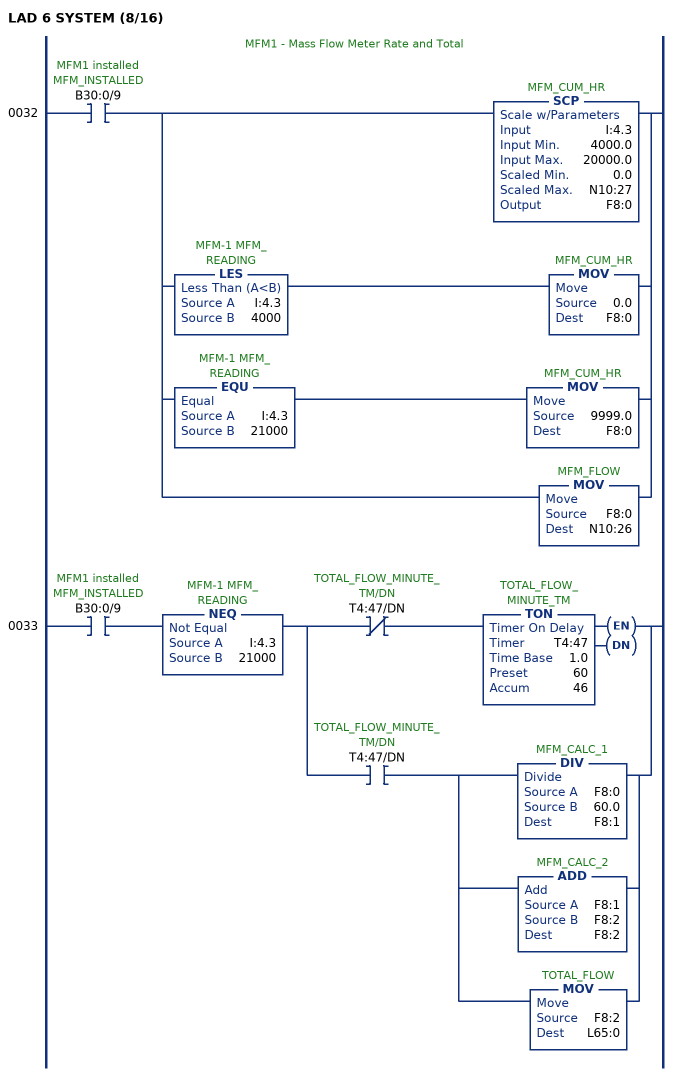
% Rung: 32 %
% MFM1 - Mass Flow Meter Rate and Total %
SOR XIC B30:0/9 BST SCP I:4.3 4000.0 20000.0 0.0 N10:27 F8:0 NXB LES I:4.3 4000 MOV 0.0 F8:0 NXB EQU I:4.3 21000 MOV 9999.0 F8:0 NXB MOV F8:0 N10:26 BND EOR
%   B30:0/9  MFM_INSTALLED  "MFM1 installed" %
%   I:4.3  MFM_READING  "MFM-1" %
%   N10:27  MFM_SCALING %
%   F8:0  MFM_CUM_HR %
%   N10:26  MFM_FLOW %
% Rung: 33 %
SOR XIC B30:0/9 NEQ I:4.3 21000 BST XIO T4:47/DN TON T4:47 1.0 60 46 NXB XIC T4:47/DN BST DIV F8:0 60.0 F8:1 NXB ADD F8:1 F8:2 F8:2 NXB MOV F8:2 L65:0 BND BND EOR
%   B30:0/9  MFM_INSTALLED  "MFM1 installed" %
%   I:4.3  MFM_READING  "MFM-1" %
%   T4:47  TOTAL_FLOW_MINUTE_TM %
%   F8:0  MFM_CUM_HR %
%   F8:1  MFM_CALC_1 %
%   F8:2  MFM_CALC_2 %
%   L65:0  TOTAL_FLOW %

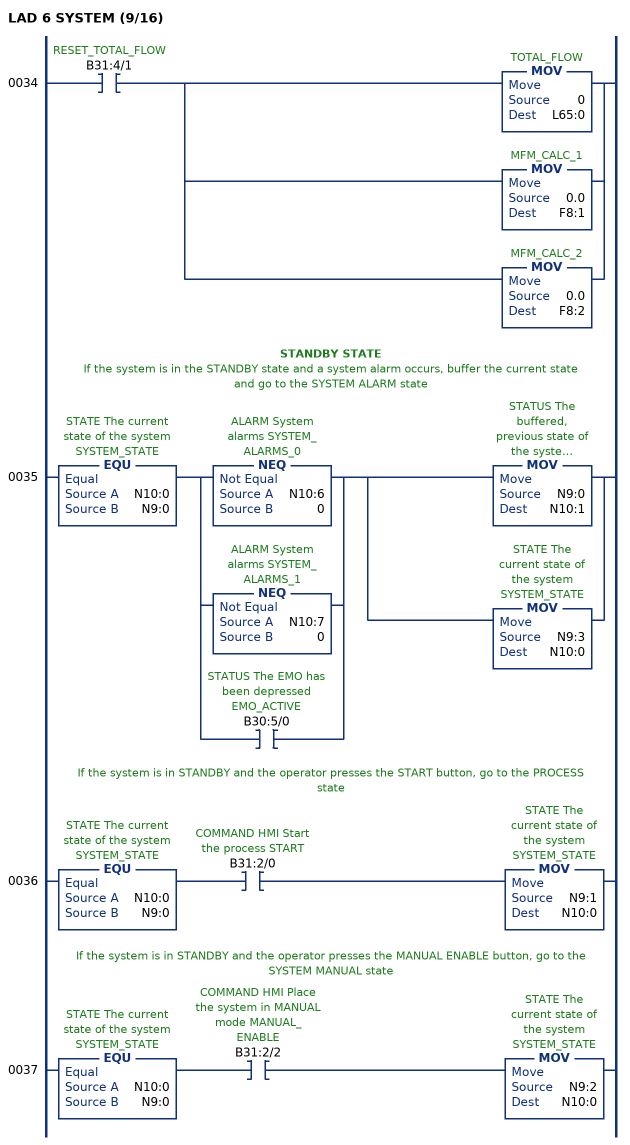
% Rung: 34 %
SOR XIC B31:4/1 BST MOV 0 L65:0 NXB MOV 0.0 F8:1 NXB MOV 0.0 F8:2 BND EOR
%   B31:4/1  RESET_TOTAL_FLOW %
%   L65:0  TOTAL_FLOW %
%   F8:1  MFM_CALC_1 %
%   F8:2  MFM_CALC_2 %
% Rung: 35 %
% TITLE: STANDBY STATE %
% If the system is in the STANDBY state and a system alarm occurs, buffer the current state and go to the SYSTEM ALARM state %
SOR EQU N10:0 N9:0 BST NEQ N10:6 0 NXB NEQ N10:7 0 NXB XIC B30:5/0 BND BST MOV N9:0 N10:1 NXB MOV N9:3 N10:0 BND EOR
%   N10:0  SYSTEM_STATE  "STATE The current state of the system" %
%   N9:0  SYSTEM_STANDBY  "STATE System Standby" %
%   N10:6  SYSTEM_ALARMS_0  "ALARM System alarms" %
%   N10:7  SYSTEM_ALARMS_1  "ALARM System alarms" %
%   B30:5/0  EMO_ACTIVE  "STATUS The EMO has been depressed" %
%   N10:1  SYSTEM_BUFFER  "STATUS The buffered, previous state of the system" %
%   N9:3  SYSTEM_ALARM  "STATE System Alarm" %
% Rung: 36 %
% If the system is in STANDBY and the operator presses the START button, go to the PROCESS state %
SOR EQU N10:0 N9:0 XIC B31:2/0 MOV N9:1 N10:0 EOR
%   N10:0  SYSTEM_STATE  "STATE The current state of the system" %
%   N9:0  SYSTEM_STANDBY  "STATE System Standby" %
%   B31:2/0  START  "COMMAND HMI Start the process" %
%   N9:1  SYSTEM_PROCESS  "STATE System Process" %
% Rung: 37 %
% If the system is in STANDBY and the operator presses the MANUAL ENABLE button, go to the SYSTEM MANUAL state %
SOR EQU N10:0 N9:0 XIC B31:2/2 MOV N9:2 N10:0 EOR
%   N10:0  SYSTEM_STATE  "STATE The current state of the system" %
%   N9:0  SYSTEM_STANDBY  "STATE System Standby" %
%   B31:2/2  MANUAL_ENABLE  "COMMAND HMI Place the system in MANUAL mode" %
%   N9:2  SYSTEM_MANUAL  "STATE System Manual" %

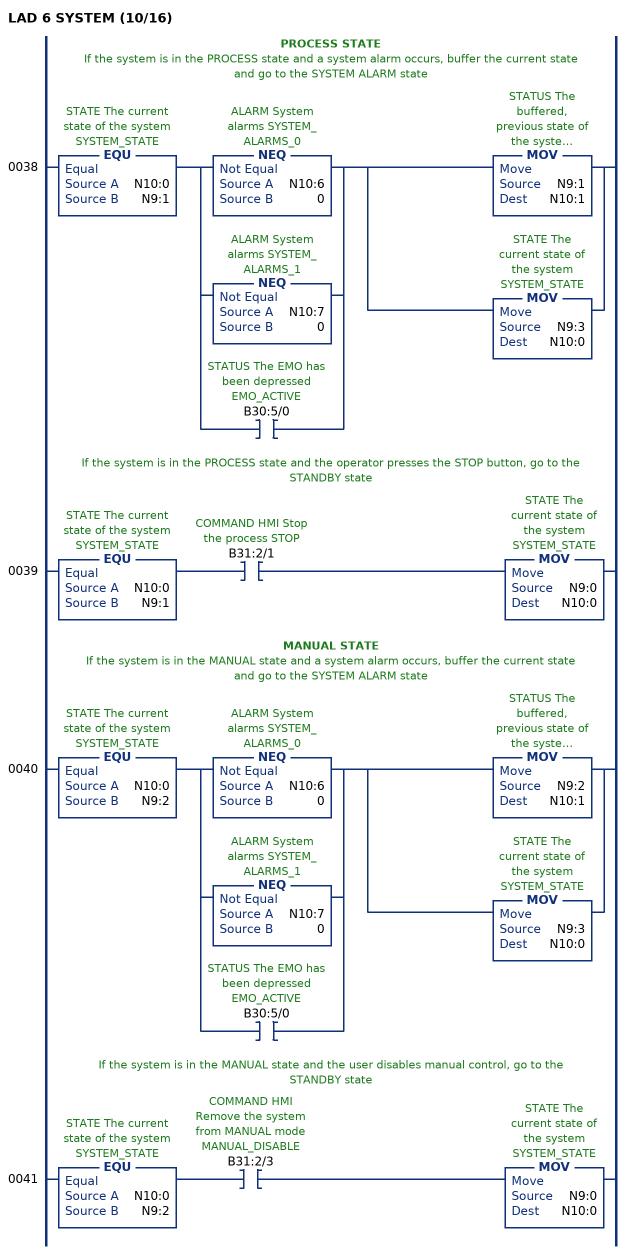
% Rung: 38 %
% TITLE: PROCESS STATE %
% If the system is in the PROCESS state and a system alarm occurs, buffer the current state and go to the SYSTEM ALARM state %
SOR EQU N10:0 N9:1 BST NEQ N10:6 0 NXB NEQ N10:7 0 NXB XIC B30:5/0 BND BST MOV N9:1 N10:1 NXB MOV N9:3 N10:0 BND EOR
%   N10:0  SYSTEM_STATE  "STATE The current state of the system" %
%   N9:1  SYSTEM_PROCESS  "STATE System Process" %
%   N10:6  SYSTEM_ALARMS_0  "ALARM System alarms" %
%   N10:7  SYSTEM_ALARMS_1  "ALARM System alarms" %
%   B30:5/0  EMO_ACTIVE  "STATUS The EMO has been depressed" %
%   N10:1  SYSTEM_BUFFER  "STATUS The buffered, previous state of the system" %
%   N9:3  SYSTEM_ALARM  "STATE System Alarm" %
% Rung: 39 %
% If the system is in the PROCESS state and the operator presses the STOP button, go to the STANDBY state %
SOR EQU N10:0 N9:1 XIC B31:2/1 MOV N9:0 N10:0 EOR
%   N10:0  SYSTEM_STATE  "STATE The current state of the system" %
%   N9:1  SYSTEM_PROCESS  "STATE System Process" %
%   B31:2/1  STOP  "COMMAND HMI Stop the process" %
%   N9:0  SYSTEM_STANDBY  "STATE System Standby" %
% Rung: 40 %
% TITLE: MANUAL STATE %
% If the system is in the MANUAL state and a system alarm occurs, buffer the current state and go to the SYSTEM ALARM state %
SOR EQU N10:0 N9:2 BST NEQ N10:6 0 NXB NEQ N10:7 0 NXB XIC B30:5/0 BND BST MOV N9:2 N10:1 NXB MOV N9:3 N10:0 BND EOR
%   N10:0  SYSTEM_STATE  "STATE The current state of the system" %
%   N9:2  SYSTEM_MANUAL  "STATE System Manual" %
%   N10:6  SYSTEM_ALARMS_0  "ALARM System alarms" %
%   N10:7  SYSTEM_ALARMS_1  "ALARM System alarms" %
%   B30:5/0  EMO_ACTIVE  "STATUS The EMO has been depressed" %
%   N10:1  SYSTEM_BUFFER  "STATUS The buffered, previous state of the system" %
%   N9:3  SYSTEM_ALARM  "STATE System Alarm" %
% Rung: 41 %
% If the system is in the MANUAL state and the user disables manual control, go to the STANDBY state %
SOR EQU N10:0 N9:2 XIC B31:2/3 MOV N9:0 N10:0 EOR
%   N10:0  SYSTEM_STATE  "STATE The current state of the system" %
%   N9:2  SYSTEM_MANUAL  "STATE System Manual" %
%   B31:2/3  MANUAL_DISABLE  "COMMAND HMI Remove the system from MANUAL mode" %
%   N9:0  SYSTEM_STANDBY  "STATE System Standby" %

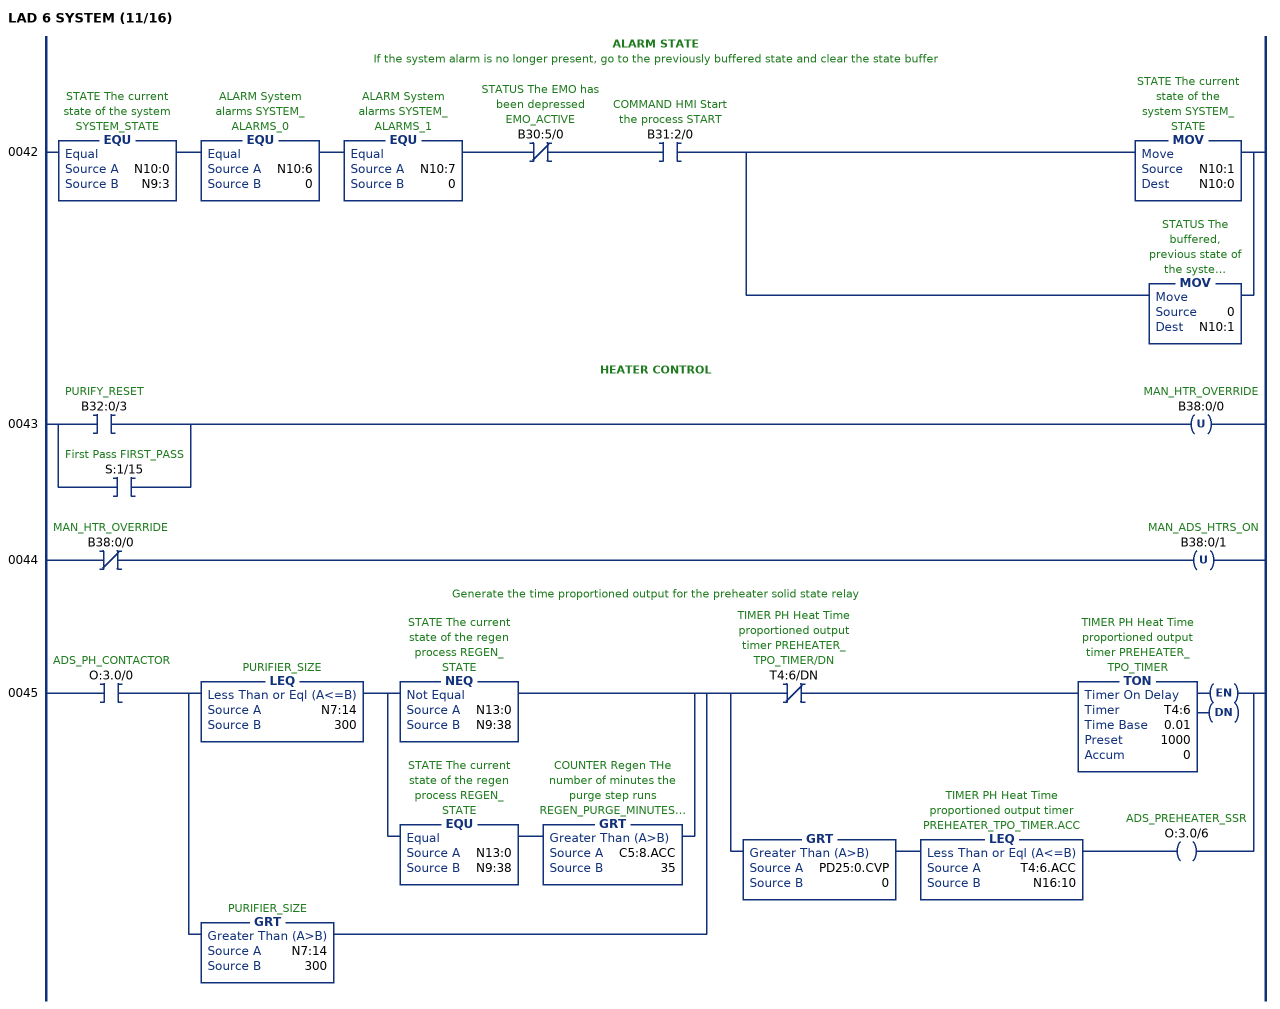
% Rung: 42 %
% TITLE: ALARM STATE %
% If the system alarm is no longer present, go to the previously buffered state and clear the state buffer %
SOR EQU N10:0 N9:3 EQU N10:6 0 EQU N10:7 0 XIO B30:5/0 XIC B31:2/0 BST MOV N10:1 N10:0 NXB MOV 0 N10:1 BND EOR
%   N10:0  SYSTEM_STATE  "STATE The current state of the system" %
%   N9:3  SYSTEM_ALARM  "STATE System Alarm" %
%   N10:6  SYSTEM_ALARMS_0  "ALARM System alarms" %
%   N10:7  SYSTEM_ALARMS_1  "ALARM System alarms" %
%   B30:5/0  EMO_ACTIVE  "STATUS The EMO has been depressed" %
%   B31:2/0  START  "COMMAND HMI Start the process" %
%   N10:1  SYSTEM_BUFFER  "STATUS The buffered, previous state of the system" %
% Rung: 43 %
% TITLE: HEATER CONTROL %
SOR BST XIC B32:0/3 NXB XIC S:1/15 BND OTU B38:0/0 EOR
%   B32:0/3  PURIFY_RESET %
%   S:1/15  FIRST_PASS  "First Pass" %
%   B38:0/0  MAN_HTR_OVERRIDE %
% Rung: 44 %
SOR XIO B38:0/0 OTU B38:0/1 EOR
%   B38:0/0  MAN_HTR_OVERRIDE %
%   B38:0/1  MAN_ADS_HTRS_ON %
% Rung: 45 %
% Generate the time proportioned output for the preheater solid state relay %
SOR XIC O:3.0/0 BST LEQ N7:14 300 BST NEQ N13:0 N9:38 NXB EQU N13:0 N9:38 GRT C5:8.ACC 35 BND NXB GRT N7:14 300 BND BST XIO T4:6/DN TON T4:6 0.01 1000 0 NXB GRT PD25:0.CVP 0 LEQ T4:6.ACC N16:10 OTE O:3.0/6 BND EOR
%   O:3.0/0  ADS_PH_CONTACTOR %
%   N7:14  PURIFIER_SIZE %
%   N13:0  REGEN_STATE  "STATE The current state of the regen process" %
%   N9:38  REGEN_PURGE  "STATE Regen Hot Purge" %
%   C5:8  REGEN_PURGE_MINUTES  "COUNTER Regen THe number of minutes the purge step runs" %
%   T4:6  PREHEATER_TPO_TIMER  "TIMER PH Heat Time proportioned output timer" %
%   N16:10  ADS_PH_OUTPUT  "CONTROL ADS Preheater output (percent)" %
%   O:3.0/6  ADS_PREHEATER_SSR %

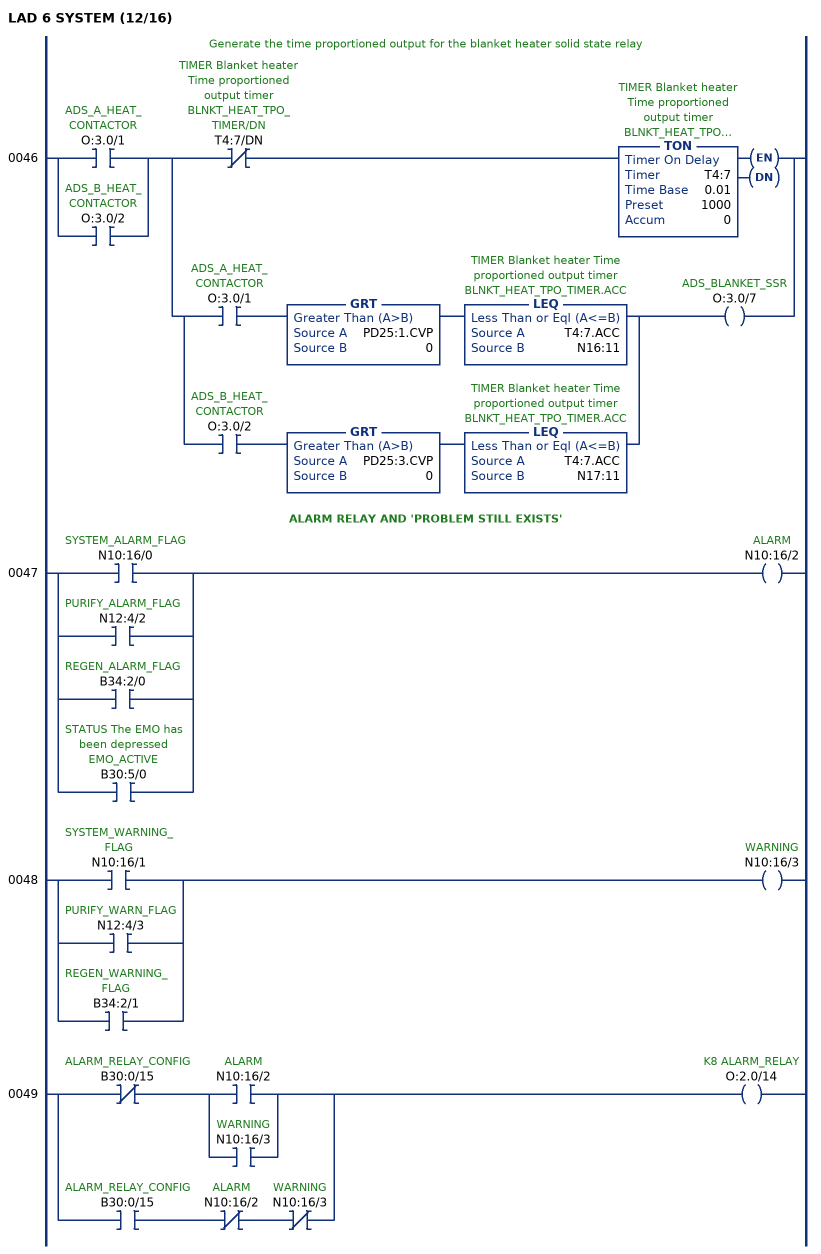
% Rung: 46 %
% Generate the time proportioned output for the blanket heater solid state relay %
SOR BST XIC O:3.0/1 NXB XIC O:3.0/2 BND BST XIO T4:7/DN TON T4:7 0.01 1000 0 NXB BST XIC O:3.0/1 GRT PD25:1.CVP 0 LEQ T4:7.ACC N16:11 NXB XIC O:3.0/2 GRT PD25:3.CVP 0 LEQ T4:7.ACC N17:11 BND OTE O:3.0/7 BND EOR
%   O:3.0/1  ADS_A_HEAT_CONTACTOR %
%   O:3.0/2  ADS_B_HEAT_CONTACTOR %
%   T4:7  BLNKT_HEAT_TPO_TIMER  "TIMER Blanket heater Time proportioned output timer" %
%   N16:11  ADS_A_BLNKT_OUTPUT  "CONTROL ADS A Blanket output (percent)" %
%   N17:11  ADS_B_BLNKT_OUTPUT  "CONTROL ADS A Blanket output" %
%   O:3.0/7  ADS_BLANKET_SSR %
% Rung: 47 %
% TITLE: ALARM RELAY AND 'PROBLEM STILL EXISTS' %
SOR BST XIC N10:16/0 NXB XIC N12:4/2 NXB XIC B34:2/0 NXB XIC B30:5/0 BND OTE N10:16/2 EOR
%   N10:16/0  SYSTEM_ALARM_FLAG %
%   N12:4/2  PURIFY_ALARM_FLAG %
%   B34:2/0  REGEN_ALARM_FLAG %
%   B30:5/0  EMO_ACTIVE  "STATUS The EMO has been depressed" %
%   N10:16/2  ALARM %
% Rung: 48 %
SOR BST XIC N10:16/1 NXB XIC N12:4/3 NXB XIC B34:2/1 BND OTE N10:16/3 EOR
%   N10:16/1  SYSTEM_WARNING_FLAG %
%   N12:4/3  PURIFY_WARN_FLAG %
%   B34:2/1  REGEN_WARNING_FLAG %
%   N10:16/3  WARNING %
% Rung: 49 %
SOR BST XIO B30:0/15 BST XIC N10:16/2 NXB XIC N10:16/3 BND NXB XIC B30:0/15 XIO N10:16/2 XIO N10:16/3 BND OTE O:2.0/14 EOR
%   B30:0/15  ALARM_RELAY_CONFIG %
%   N10:16/2  ALARM %
%   N10:16/3  WARNING %
%   O:2.0/14  ALARM_RELAY  "K8" %

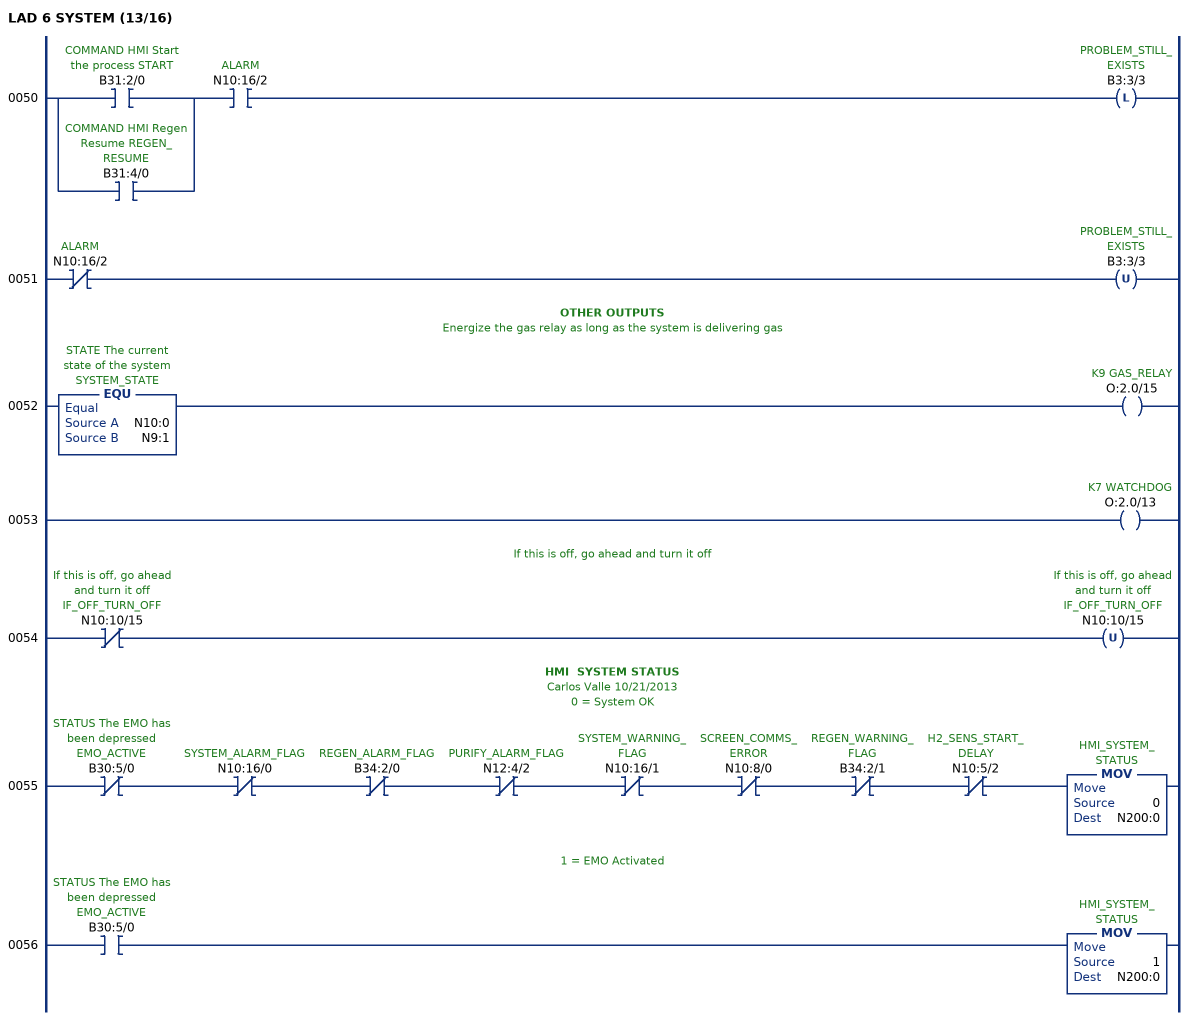
% Rung: 50 %
SOR BST XIC B31:2/0 NXB XIC B31:4/0 BND XIC N10:16/2 OTL B3:3/3 EOR
%   B31:2/0  START  "COMMAND HMI Start the process" %
%   B31:4/0  REGEN_RESUME  "COMMAND HMI Regen Resume" %
%   N10:16/2  ALARM %
%   B3:3/3  PROBLEM_STILL_EXISTS %
% Rung: 51 %
SOR XIO N10:16/2 OTU B3:3/3 EOR
%   N10:16/2  ALARM %
%   B3:3/3  PROBLEM_STILL_EXISTS %
% Rung: 52 %
% TITLE: OTHER OUTPUTS %
% Energize the gas relay as long as the system is delivering gas %
SOR EQU N10:0 N9:1 OTE O:2.0/15 EOR
%   N10:0  SYSTEM_STATE  "STATE The current state of the system" %
%   N9:1  SYSTEM_PROCESS  "STATE System Process" %
%   O:2.0/15  GAS_RELAY  "K9" %
% Rung: 53 %
SOR OTE O:2.0/13 EOR
%   O:2.0/13  WATCHDOG  "K7" %
% Rung: 54 %
% If this is off, go ahead and turn it off %
SOR XIO N10:10/15 OTU N10:10/15 EOR
%   N10:10/15  IF_OFF_TURN_OFF  "If this is off, go ahead and turn it off" %
% Rung: 55 %
% TITLE: HMI  SYSTEM STATUS %
% Carlos Valle 10/21/2013
% 0 = System OK %
SOR XIO B30:5/0 XIO N10:16/0 XIO B34:2/0 XIO N12:4/2 XIO N10:16/1 XIO N10:8/0 XIO B34:2/1 XIO N10:5/2 MOV 0 N200:0 EOR
%   B30:5/0  EMO_ACTIVE  "STATUS The EMO has been depressed" %
%   N10:16/0  SYSTEM_ALARM_FLAG %
%   B34:2/0  REGEN_ALARM_FLAG %
%   N12:4/2  PURIFY_ALARM_FLAG %
%   N10:16/1  SYSTEM_WARNING_FLAG %
%   N10:8/0  SCREEN_COMMS_ERROR %
%   B34:2/1  REGEN_WARNING_FLAG %
%   N10:5/2  H2_SENS_START_DELAY %
%   N200:0  HMI_SYSTEM_STATUS %
% Rung: 56 %
% 1 = EMO Activated %
SOR XIC B30:5/0 MOV 1 N200:0 EOR
%   B30:5/0  EMO_ACTIVE  "STATUS The EMO has been depressed" %
%   N200:0  HMI_SYSTEM_STATUS %

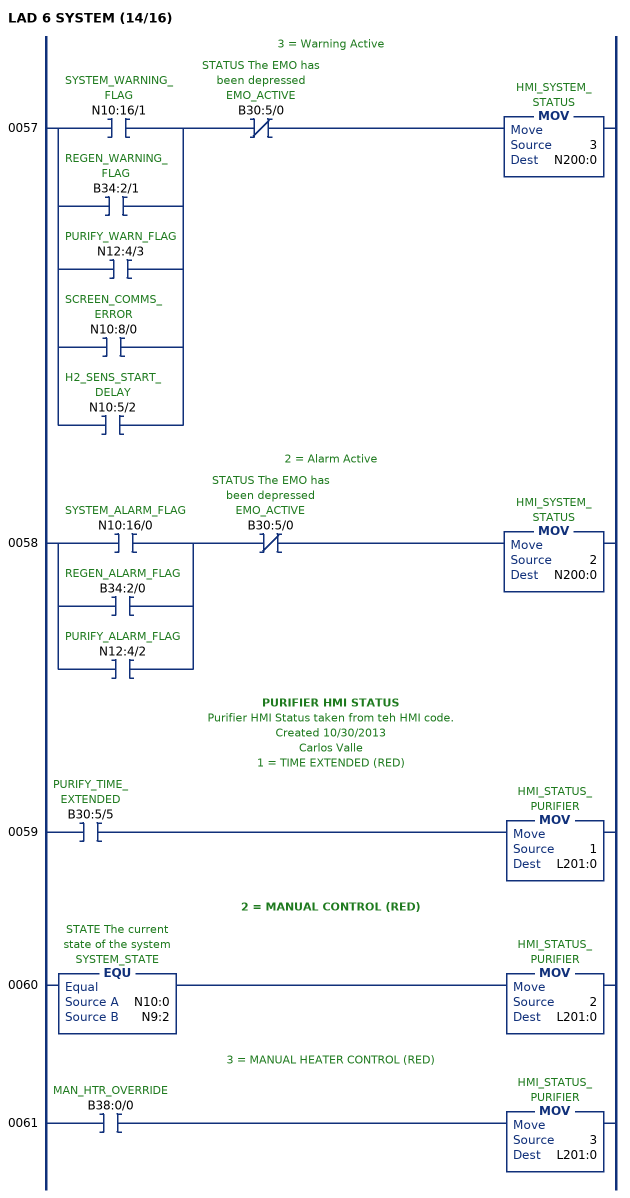
% Rung: 57 %
% 3 = Warning Active %
SOR BST XIC N10:16/1 NXB XIC B34:2/1 NXB XIC N12:4/3 NXB XIC N10:8/0 NXB XIC N10:5/2 BND XIO B30:5/0 MOV 3 N200:0 EOR
%   N10:16/1  SYSTEM_WARNING_FLAG %
%   B34:2/1  REGEN_WARNING_FLAG %
%   N12:4/3  PURIFY_WARN_FLAG %
%   N10:8/0  SCREEN_COMMS_ERROR %
%   N10:5/2  H2_SENS_START_DELAY %
%   B30:5/0  EMO_ACTIVE  "STATUS The EMO has been depressed" %
%   N200:0  HMI_SYSTEM_STATUS %
% Rung: 58 %
% 2 = Alarm Active %
SOR BST XIC N10:16/0 NXB XIC B34:2/0 NXB XIC N12:4/2 BND XIO B30:5/0 MOV 2 N200:0 EOR
%   N10:16/0  SYSTEM_ALARM_FLAG %
%   B34:2/0  REGEN_ALARM_FLAG %
%   N12:4/2  PURIFY_ALARM_FLAG %
%   B30:5/0  EMO_ACTIVE  "STATUS The EMO has been depressed" %
%   N200:0  HMI_SYSTEM_STATUS %
% Rung: 59 %
% TITLE: PURIFIER HMI STATUS %
% Purifier HMI Status taken from teh HMI code.
% Created 10/30/2013
% Carlos Valle
% 1 = TIME EXTENDED (RED) %
SOR XIC B30:5/5 MOV 1 L201:0 EOR
%   B30:5/5  PURIFY_TIME_EXTENDED %
%   L201:0  HMI_STATUS_PURIFIER %
% Rung: 60 %
% TITLE: 2 = MANUAL CONTROL (RED) %
SOR EQU N10:0 N9:2 MOV 2 L201:0 EOR
%   N10:0  SYSTEM_STATE  "STATE The current state of the system" %
%   N9:2  SYSTEM_MANUAL  "STATE System Manual" %
%   L201:0  HMI_STATUS_PURIFIER %
% Rung: 61 %
% 3 = MANUAL HEATER CONTROL (RED) %
SOR XIC B38:0/0 MOV 3 L201:0 EOR
%   B38:0/0  MAN_HTR_OVERRIDE %
%   L201:0  HMI_STATUS_PURIFIER %

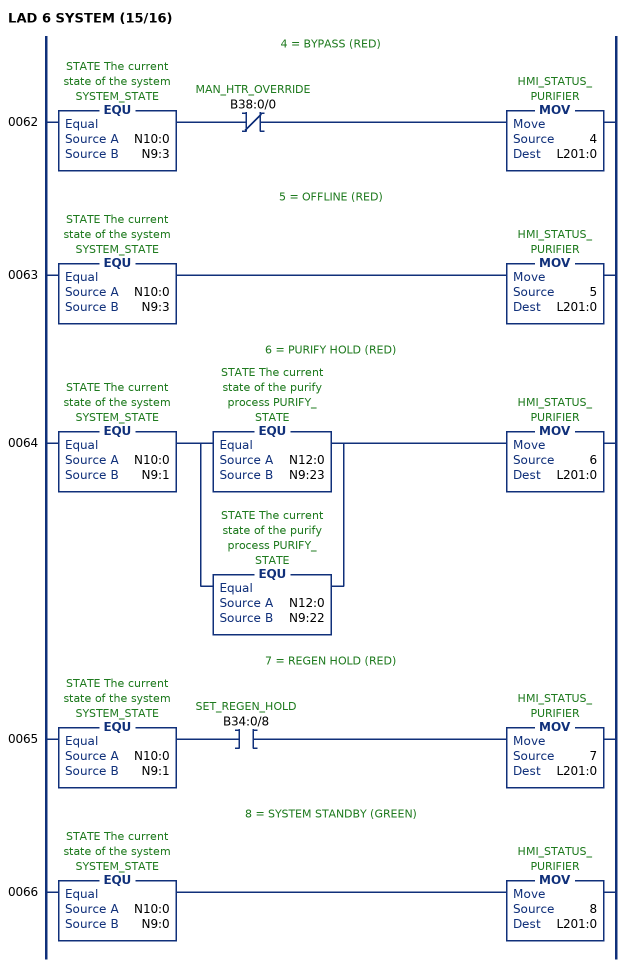
% Rung: 62 %
% 4 = BYPASS (RED) %
SOR EQU N10:0 N9:3 XIO B38:0/0 MOV 4 L201:0 EOR
%   N10:0  SYSTEM_STATE  "STATE The current state of the system" %
%   N9:3  SYSTEM_ALARM  "STATE System Alarm" %
%   B38:0/0  MAN_HTR_OVERRIDE %
%   L201:0  HMI_STATUS_PURIFIER %
% Rung: 63 %
% 5 = OFFLINE (RED) %
SOR EQU N10:0 N9:3 MOV 5 L201:0 EOR
%   N10:0  SYSTEM_STATE  "STATE The current state of the system" %
%   N9:3  SYSTEM_ALARM  "STATE System Alarm" %
%   L201:0  HMI_STATUS_PURIFIER %
% Rung: 64 %
% 6 = PURIFY HOLD (RED) %
SOR EQU N10:0 N9:1 BST EQU N12:0 N9:23 NXB EQU N12:0 N9:22 BND MOV 6 L201:0 EOR
%   N10:0  SYSTEM_STATE  "STATE The current state of the system" %
%   N9:1  SYSTEM_PROCESS  "STATE System Process" %
%   N12:0  PURIFY_STATE  "STATE The current state of the purify process" %
%   N9:23  PURIFY_MANUAL_HOLD  "STATE Purify Manual Hold" %
%   N9:22  PURIFY_HOLD  "STATE Purify Hold" %
%   L201:0  HMI_STATUS_PURIFIER %
% Rung: 65 %
% 7 = REGEN HOLD (RED) %
SOR EQU N10:0 N9:1 XIC B34:0/8 MOV 7 L201:0 EOR
%   N10:0  SYSTEM_STATE  "STATE The current state of the system" %
%   N9:1  SYSTEM_PROCESS  "STATE System Process" %
%   B34:0/8  SET_REGEN_HOLD %
%   L201:0  HMI_STATUS_PURIFIER %
% Rung: 66 %
% 8 = SYSTEM STANDBY (GREEN) %
SOR EQU N10:0 N9:0 MOV 8 L201:0 EOR
%   N10:0  SYSTEM_STATE  "STATE The current state of the system" %
%   N9:0  SYSTEM_STANDBY  "STATE System Standby" %
%   L201:0  HMI_STATUS_PURIFIER %

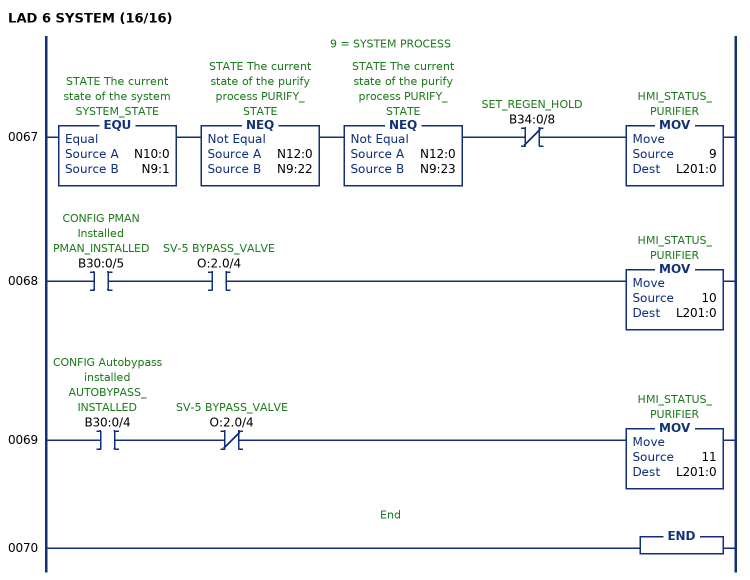
% Rung: 67 %
% 9 = SYSTEM PROCESS %
SOR EQU N10:0 N9:1 NEQ N12:0 N9:22 NEQ N12:0 N9:23 XIO B34:0/8 MOV 9 L201:0 EOR
%   N10:0  SYSTEM_STATE  "STATE The current state of the system" %
%   N9:1  SYSTEM_PROCESS  "STATE System Process" %
%   N12:0  PURIFY_STATE  "STATE The current state of the purify process" %
%   N9:22  PURIFY_HOLD  "STATE Purify Hold" %
%   N9:23  PURIFY_MANUAL_HOLD  "STATE Purify Manual Hold" %
%   B34:0/8  SET_REGEN_HOLD %
%   L201:0  HMI_STATUS_PURIFIER %
% Rung: 68 %
SOR XIC B30:0/5 XIC O:2.0/4 MOV 10 L201:0 EOR
%   B30:0/5  PMAN_INSTALLED  "CONFIG PMAN Installed" %
%   O:2.0/4  BYPASS_VALVE  "SV-5" %
%   L201:0  HMI_STATUS_PURIFIER %
% Rung: 69 %
SOR XIC B30:0/4 XIO O:2.0/4 MOV 11 L201:0 EOR
%   B30:0/4  AUTOBYPASS_INSTALLED  "CONFIG Autobypass installed" %
%   O:2.0/4  BYPASS_VALVE  "SV-5" %
%   L201:0  HMI_STATUS_PURIFIER %
% Rung: 70 %
% End %
SOR END EOR

LADDER 7 "PROCESSING"    % Runs the processing control %
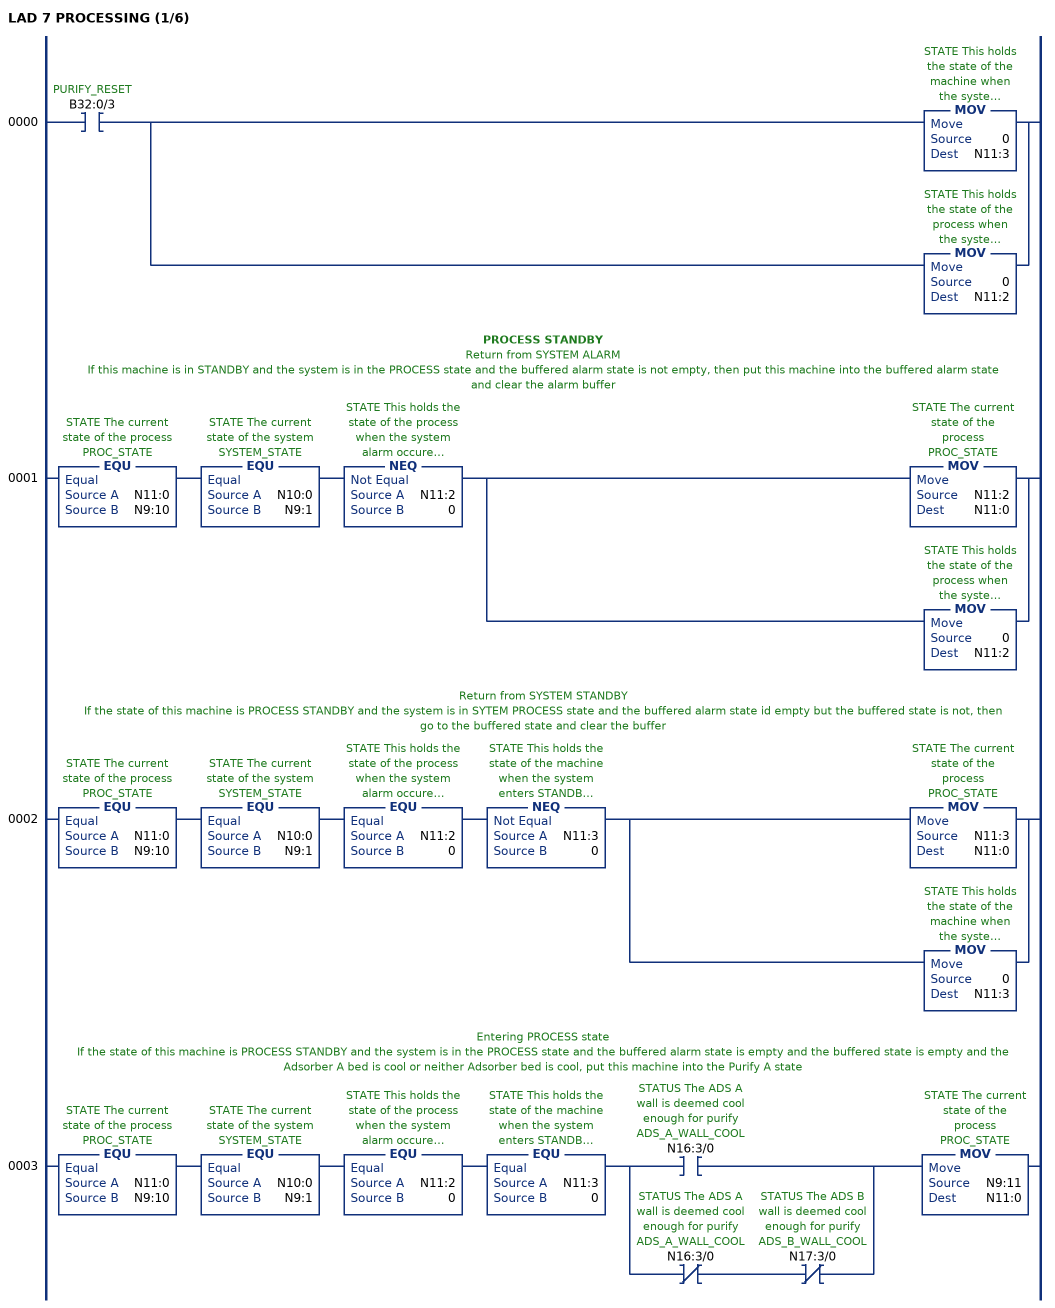
% Rung: 0 %
SOR XIC B32:0/3 BST MOV 0 N11:3 NXB MOV 0 N11:2 BND EOR
%   B32:0/3  PURIFY_RESET %
%   N11:3  PROC_STANDBY_BUFFER  "STATE This holds the state of the machine when the system enters STANDBY state" %
%   N11:2  PROC_ALARM_BUFFER  "STATE This holds the state of the process when the system alarm occured" %
% Rung: 1 %
% TITLE: PROCESS STANDBY %
% Return from SYSTEM ALARM
% If this machine is in STANDBY and the system is in the PROCESS state and the buffered alarm state is not empty, then put this machine into the buffered alarm state and clear the alarm buffer %
SOR EQU N11:0 N9:10 EQU N10:0 N9:1 NEQ N11:2 0 BST MOV N11:2 N11:0 NXB MOV 0 N11:2 BND EOR
%   N11:0  PROC_STATE  "STATE The current state of the process" %
%   N9:10  PROC_STANDBY  "STATE Process Standby" %
%   N10:0  SYSTEM_STATE  "STATE The current state of the system" %
%   N9:1  SYSTEM_PROCESS  "STATE System Process" %
%   N11:2  PROC_ALARM_BUFFER  "STATE This holds the state of the process when the system alarm occured" %
% Rung: 2 %
% Return from SYSTEM STANDBY
% If the state of this machine is PROCESS STANDBY and the system is in SYTEM PROCESS state and the buffered alarm state id empty but the buffered state is not, then go to the buffered state and clear the buffer %
SOR EQU N11:0 N9:10 EQU N10:0 N9:1 EQU N11:2 0 NEQ N11:3 0 BST MOV N11:3 N11:0 NXB MOV 0 N11:3 BND EOR
%   N11:0  PROC_STATE  "STATE The current state of the process" %
%   N9:10  PROC_STANDBY  "STATE Process Standby" %
%   N10:0  SYSTEM_STATE  "STATE The current state of the system" %
%   N9:1  SYSTEM_PROCESS  "STATE System Process" %
%   N11:2  PROC_ALARM_BUFFER  "STATE This holds the state of the process when the system alarm occured" %
%   N11:3  PROC_STANDBY_BUFFER  "STATE This holds the state of the machine when the system enters STANDBY state" %
% Rung: 3 %
% Entering PROCESS state
% If the state of this machine is PROCESS STANDBY and the system is in the PROCESS state and the buffered alarm state is empty and the buffered state is empty and the Adsorber A bed is cool or neither Adsorber bed is cool, put this machine into the Purify A state %
SOR EQU N11:0 N9:10 EQU N10:0 N9:1 EQU N11:2 0 EQU N11:3 0 BST XIC N16:3/0 NXB XIO N16:3/0 XIO N17:3/0 BND MOV N9:11 N11:0 EOR
%   N11:0  PROC_STATE  "STATE The current state of the process" %
%   N9:10  PROC_STANDBY  "STATE Process Standby" %
%   N10:0  SYSTEM_STATE  "STATE The current state of the system" %
%   N9:1  SYSTEM_PROCESS  "STATE System Process" %
%   N11:2  PROC_ALARM_BUFFER  "STATE This holds the state of the process when the system alarm occured" %
%   N11:3  PROC_STANDBY_BUFFER  "STATE This holds the state of the machine when the system enters STANDBY state" %
%   N16:3/0  ADS_A_WALL_COOL  "STATUS The ADS A wall is deemed cool enough for purify" %
%   N17:3/0  ADS_B_WALL_COOL  "STATUS The ADS B wall is deemed cool enough for purify" %
%   N9:11  PROC_PURIFY_A  "STATE Process Purify A" %

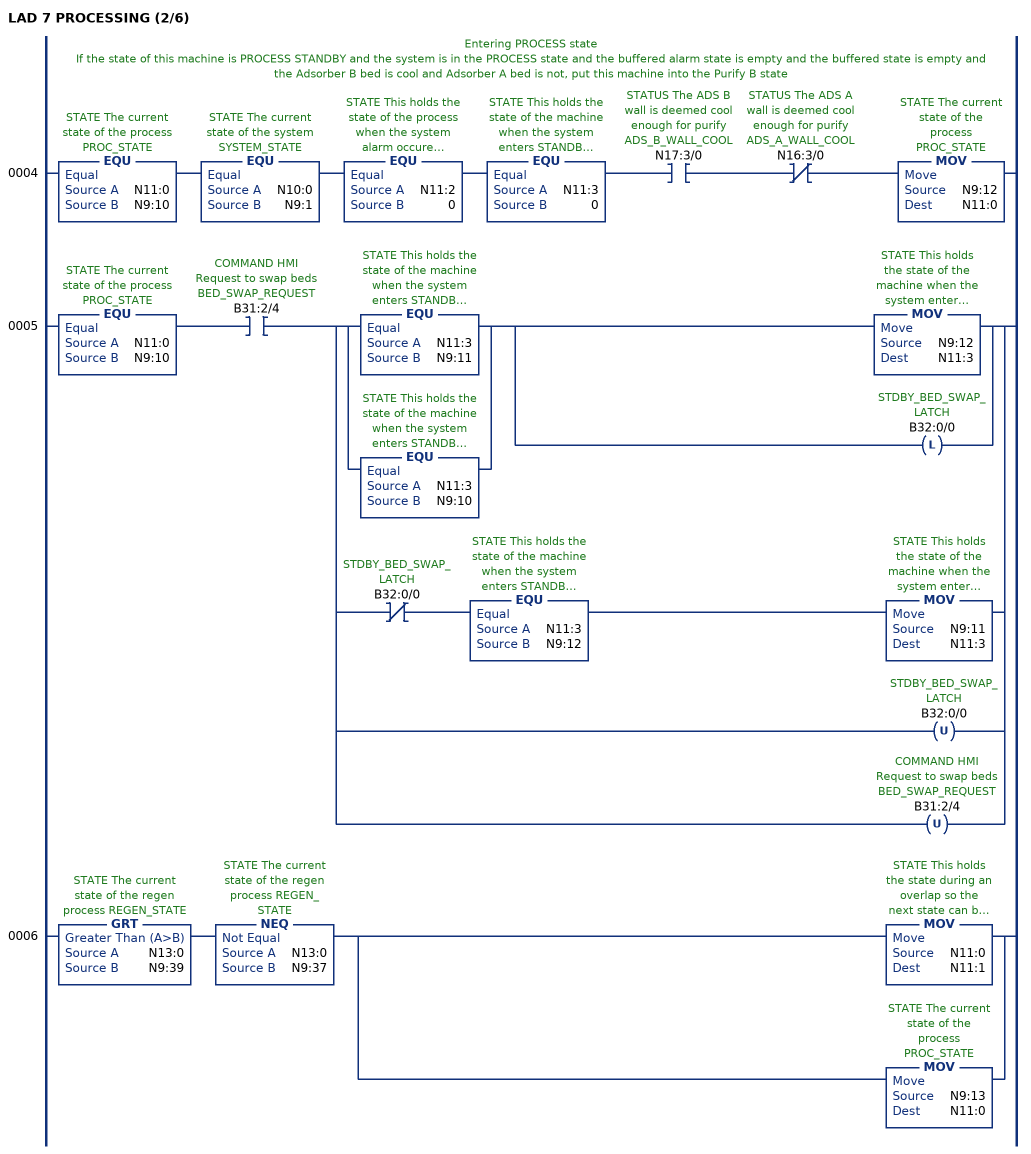
% Rung: 4 %
% Entering PROCESS state
% If the state of this machine is PROCESS STANDBY and the system is in the PROCESS state and the buffered alarm state is empty and the buffered state is empty and the Adsorber B bed is cool and Adsorber A bed is not, put this machine into the Purify B state %
SOR EQU N11:0 N9:10 EQU N10:0 N9:1 EQU N11:2 0 EQU N11:3 0 XIC N17:3/0 XIO N16:3/0 MOV N9:12 N11:0 EOR
%   N11:0  PROC_STATE  "STATE The current state of the process" %
%   N9:10  PROC_STANDBY  "STATE Process Standby" %
%   N10:0  SYSTEM_STATE  "STATE The current state of the system" %
%   N9:1  SYSTEM_PROCESS  "STATE System Process" %
%   N11:2  PROC_ALARM_BUFFER  "STATE This holds the state of the process when the system alarm occured" %
%   N11:3  PROC_STANDBY_BUFFER  "STATE This holds the state of the machine when the system enters STANDBY state" %
%   N17:3/0  ADS_B_WALL_COOL  "STATUS The ADS B wall is deemed cool enough for purify" %
%   N16:3/0  ADS_A_WALL_COOL  "STATUS The ADS A wall is deemed cool enough for purify" %
%   N9:12  PROC_PURIFY_B  "STATE Process Purify B" %
% Rung: 5 %
SOR EQU N11:0 N9:10 XIC B31:2/4 BST BST EQU N11:3 N9:11 NXB EQU N11:3 N9:10 BND BST MOV N9:12 N11:3 NXB OTL B32:0/0 BND NXB XIO B32:0/0 EQU N11:3 N9:12 MOV N9:11 N11:3 NXB OTU B32:0/0 NXB OTU B31:2/4 BND EOR
%   N11:0  PROC_STATE  "STATE The current state of the process" %
%   N9:10  PROC_STANDBY  "STATE Process Standby" %
%   B31:2/4  BED_SWAP_REQUEST  "COMMAND HMI Request to swap beds" %
%   N11:3  PROC_STANDBY_BUFFER  "STATE This holds the state of the machine when the system enters STANDBY state" %
%   N9:11  PROC_PURIFY_A  "STATE Process Purify A" %
%   N9:12  PROC_PURIFY_B  "STATE Process Purify B" %
%   B32:0/0  STDBY_BED_SWAP_LATCH %
% Rung: 6 %
SOR GRT N13:0 N9:39 NEQ N13:0 N9:37 BST MOV N11:0 N11:1 NXB MOV N9:13 N11:0 BND EOR
%   N13:0  REGEN_STATE  "STATE The current state of the regen process" %
%   N9:39  REGEN_EQUALIZE %
%   N9:37  REGEN_ALARM  "STATE Regen Alarm" %
%   N11:0  PROC_STATE  "STATE The current state of the process" %
%   N11:1  PROC_OVERLAP_BUFFER  "STATE This holds the state during an overlap so the next state can be determined" %
%   N9:13  PROC_OVERLAP  "STATE Process Purify Overlap" %

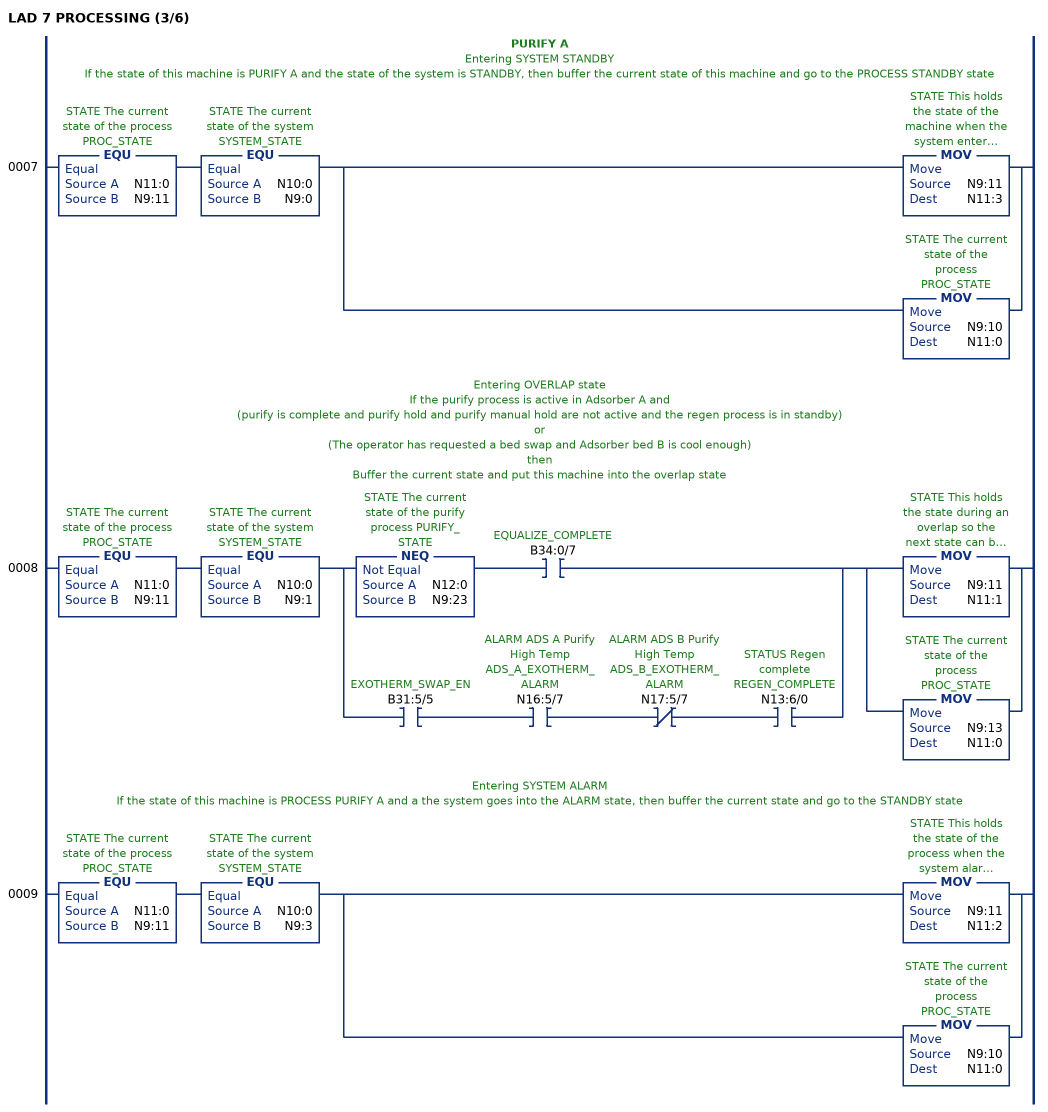
% Rung: 7 %
% TITLE: PURIFY A %
% Entering SYSTEM STANDBY
% If the state of this machine is PURIFY A and the state of the system is STANDBY, then buffer the current state of this machine and go to the PROCESS STANDBY state %
SOR EQU N11:0 N9:11 EQU N10:0 N9:0 BST MOV N9:11 N11:3 NXB MOV N9:10 N11:0 BND EOR
%   N11:0  PROC_STATE  "STATE The current state of the process" %
%   N9:11  PROC_PURIFY_A  "STATE Process Purify A" %
%   N10:0  SYSTEM_STATE  "STATE The current state of the system" %
%   N9:0  SYSTEM_STANDBY  "STATE System Standby" %
%   N11:3  PROC_STANDBY_BUFFER  "STATE This holds the state of the machine when the system enters STANDBY state" %
%   N9:10  PROC_STANDBY  "STATE Process Standby" %
% Rung: 8 %
% Entering OVERLAP state
% If the purify process is active in Adsorber A and
% (purify is complete and purify hold and purify manual hold are not active and the regen process is in standby)
% or
% (The operator has requested a bed swap and Adsorber bed B is cool enough)
% then
% Buffer the current state and put this machine into the overlap state %
SOR EQU N11:0 N9:11 EQU N10:0 N9:1 BST NEQ N12:0 N9:23 XIC B34:0/7 NXB XIC B31:5/5 XIC N16:5/7 XIO N17:5/7 XIC N13:6/0 BND BST MOV N9:11 N11:1 NXB MOV N9:13 N11:0 BND EOR
%   N11:0  PROC_STATE  "STATE The current state of the process" %
%   N9:11  PROC_PURIFY_A  "STATE Process Purify A" %
%   N10:0  SYSTEM_STATE  "STATE The current state of the system" %
%   N9:1  SYSTEM_PROCESS  "STATE System Process" %
%   N12:0  PURIFY_STATE  "STATE The current state of the purify process" %
%   N9:23  PURIFY_MANUAL_HOLD  "STATE Purify Manual Hold" %
%   B34:0/7  EQUALIZE_COMPLETE %
%   B31:5/5  EXOTHERM_SWAP_EN %
%   N16:5/7  ADS_A_EXOTHERM_ALARM  "ALARM ADS A Purify High Temp" %
%   N17:5/7  ADS_B_EXOTHERM_ALARM  "ALARM ADS B Purify High Temp" %
%   N13:6/0  REGEN_COMPLETE  "STATUS Regen complete" %
%   N11:1  PROC_OVERLAP_BUFFER  "STATE This holds the state during an overlap so the next state can be determined" %
%   N9:13  PROC_OVERLAP  "STATE Process Purify Overlap" %
% Rung: 9 %
% Entering SYSTEM ALARM
% If the state of this machine is PROCESS PURIFY A and a the system goes into the ALARM state, then buffer the current state and go to the STANDBY state %
SOR EQU N11:0 N9:11 EQU N10:0 N9:3 BST MOV N9:11 N11:2 NXB MOV N9:10 N11:0 BND EOR
%   N11:0  PROC_STATE  "STATE The current state of the process" %
%   N9:11  PROC_PURIFY_A  "STATE Process Purify A" %
%   N10:0  SYSTEM_STATE  "STATE The current state of the system" %
%   N9:3  SYSTEM_ALARM  "STATE System Alarm" %
%   N11:2  PROC_ALARM_BUFFER  "STATE This holds the state of the process when the system alarm occured" %
%   N9:10  PROC_STANDBY  "STATE Process Standby" %

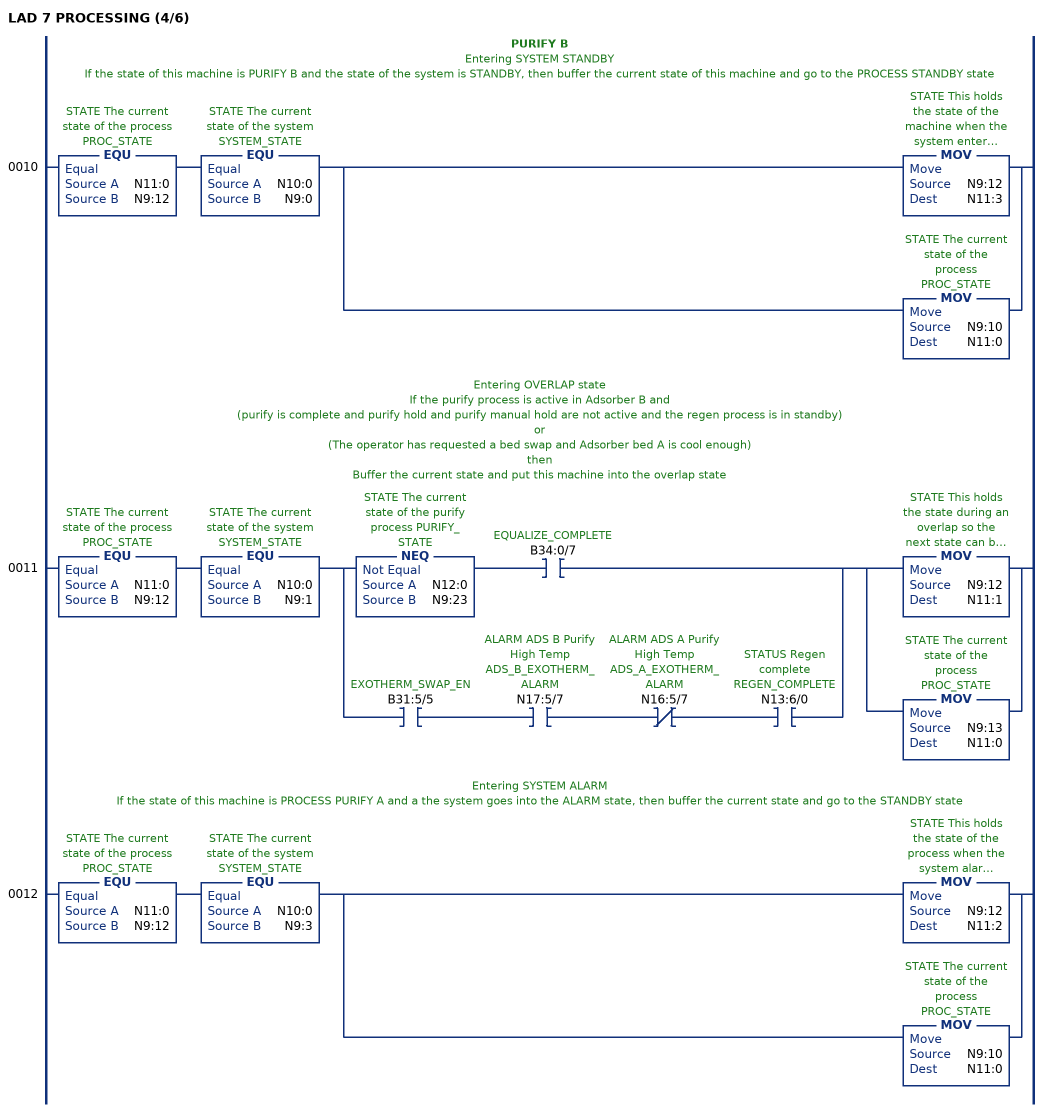
% Rung: 10 %
% TITLE: PURIFY B %
% Entering SYSTEM STANDBY
% If the state of this machine is PURIFY B and the state of the system is STANDBY, then buffer the current state of this machine and go to the PROCESS STANDBY state %
SOR EQU N11:0 N9:12 EQU N10:0 N9:0 BST MOV N9:12 N11:3 NXB MOV N9:10 N11:0 BND EOR
%   N11:0  PROC_STATE  "STATE The current state of the process" %
%   N9:12  PROC_PURIFY_B  "STATE Process Purify B" %
%   N10:0  SYSTEM_STATE  "STATE The current state of the system" %
%   N9:0  SYSTEM_STANDBY  "STATE System Standby" %
%   N11:3  PROC_STANDBY_BUFFER  "STATE This holds the state of the machine when the system enters STANDBY state" %
%   N9:10  PROC_STANDBY  "STATE Process Standby" %
% Rung: 11 %
% Entering OVERLAP state
% If the purify process is active in Adsorber B and
% (purify is complete and purify hold and purify manual hold are not active and the regen process is in standby)
% or
% (The operator has requested a bed swap and Adsorber bed A is cool enough)
% then
% Buffer the current state and put this machine into the overlap state %
SOR EQU N11:0 N9:12 EQU N10:0 N9:1 BST NEQ N12:0 N9:23 XIC B34:0/7 NXB XIC B31:5/5 XIC N17:5/7 XIO N16:5/7 XIC N13:6/0 BND BST MOV N9:12 N11:1 NXB MOV N9:13 N11:0 BND EOR
%   N11:0  PROC_STATE  "STATE The current state of the process" %
%   N9:12  PROC_PURIFY_B  "STATE Process Purify B" %
%   N10:0  SYSTEM_STATE  "STATE The current state of the system" %
%   N9:1  SYSTEM_PROCESS  "STATE System Process" %
%   N12:0  PURIFY_STATE  "STATE The current state of the purify process" %
%   N9:23  PURIFY_MANUAL_HOLD  "STATE Purify Manual Hold" %
%   B34:0/7  EQUALIZE_COMPLETE %
%   B31:5/5  EXOTHERM_SWAP_EN %
%   N17:5/7  ADS_B_EXOTHERM_ALARM  "ALARM ADS B Purify High Temp" %
%   N16:5/7  ADS_A_EXOTHERM_ALARM  "ALARM ADS A Purify High Temp" %
%   N13:6/0  REGEN_COMPLETE  "STATUS Regen complete" %
%   N11:1  PROC_OVERLAP_BUFFER  "STATE This holds the state during an overlap so the next state can be determined" %
%   N9:13  PROC_OVERLAP  "STATE Process Purify Overlap" %
% Rung: 12 %
% Entering SYSTEM ALARM
% If the state of this machine is PROCESS PURIFY A and a the system goes into the ALARM state, then buffer the current state and go to the STANDBY state %
SOR EQU N11:0 N9:12 EQU N10:0 N9:3 BST MOV N9:12 N11:2 NXB MOV N9:10 N11:0 BND EOR
%   N11:0  PROC_STATE  "STATE The current state of the process" %
%   N9:12  PROC_PURIFY_B  "STATE Process Purify B" %
%   N10:0  SYSTEM_STATE  "STATE The current state of the system" %
%   N9:3  SYSTEM_ALARM  "STATE System Alarm" %
%   N11:2  PROC_ALARM_BUFFER  "STATE This holds the state of the process when the system alarm occured" %
%   N9:10  PROC_STANDBY  "STATE Process Standby" %

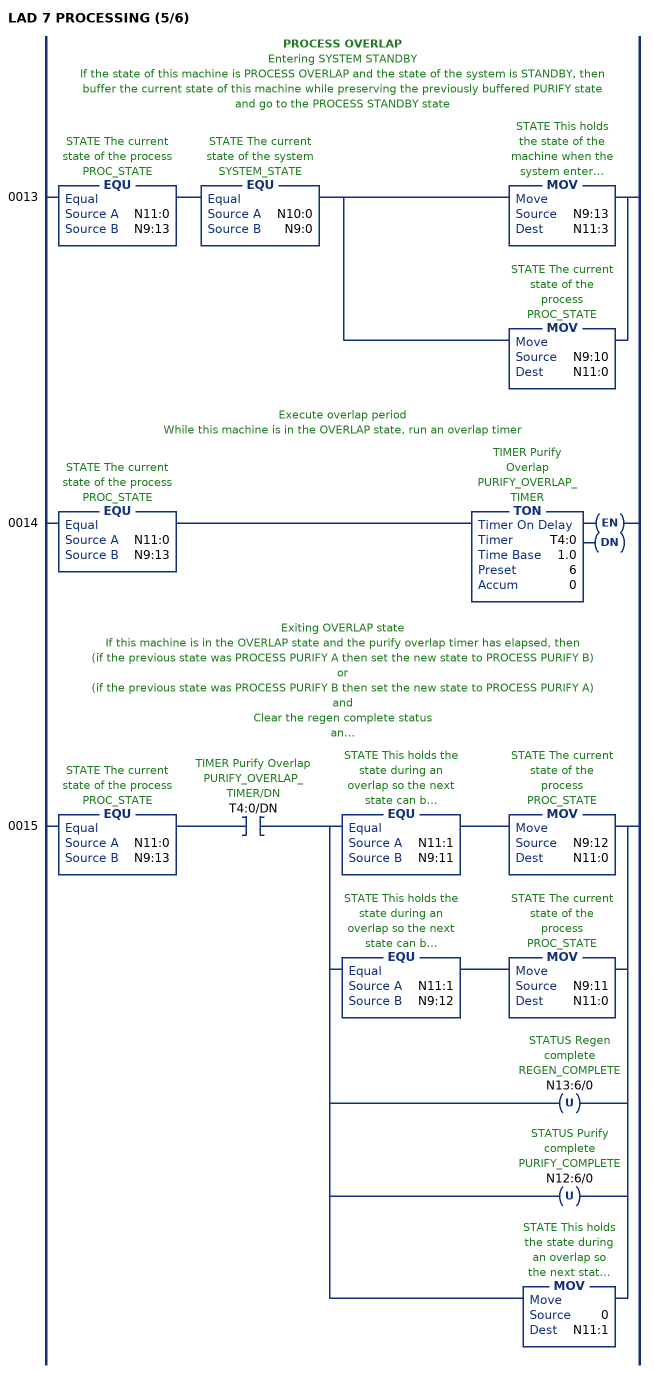
% Rung: 13 %
% TITLE: PROCESS OVERLAP %
% Entering SYSTEM STANDBY
% If the state of this machine is PROCESS OVERLAP and the state of the system is STANDBY, then buffer the current state of this machine while preserving the previously buffered PURIFY state and go to the PROCESS STANDBY state %
SOR EQU N11:0 N9:13 EQU N10:0 N9:0 BST MOV N9:13 N11:3 NXB MOV N9:10 N11:0 BND EOR
%   N11:0  PROC_STATE  "STATE The current state of the process" %
%   N9:13  PROC_OVERLAP  "STATE Process Purify Overlap" %
%   N10:0  SYSTEM_STATE  "STATE The current state of the system" %
%   N9:0  SYSTEM_STANDBY  "STATE System Standby" %
%   N11:3  PROC_STANDBY_BUFFER  "STATE This holds the state of the machine when the system enters STANDBY state" %
%   N9:10  PROC_STANDBY  "STATE Process Standby" %
% Rung: 14 %
% Execute overlap period
% While this machine is in the OVERLAP state, run an overlap timer %
SOR EQU N11:0 N9:13 TON T4:0 1.0 6 0 EOR
%   N11:0  PROC_STATE  "STATE The current state of the process" %
%   N9:13  PROC_OVERLAP  "STATE Process Purify Overlap" %
%   T4:0  PURIFY_OVERLAP_TIMER  "TIMER Purify Overlap" %
% Rung: 15 %
% Exiting OVERLAP state
% If this machine is in the OVERLAP state and the purify overlap timer has elapsed, then
% (if the previous state was PROCESS PURIFY A then set the new state to PROCESS PURIFY B)
% or
% (if the previous state was PROCESS PURIFY B then set the new state to PROCESS PURIFY A)
% and
% Clear the regen complete status
% and
% Clear the purify complete status
% and
% clear the process buffer %
SOR EQU N11:0 N9:13 XIC T4:0/DN BST EQU N11:1 N9:11 MOV N9:12 N11:0 NXB EQU N11:1 N9:12 MOV N9:11 N11:0 NXB OTU N13:6/0 NXB OTU N12:6/0 NXB MOV 0 N11:1 BND EOR
%   N11:0  PROC_STATE  "STATE The current state of the process" %
%   N9:13  PROC_OVERLAP  "STATE Process Purify Overlap" %
%   T4:0  PURIFY_OVERLAP_TIMER  "TIMER Purify Overlap" %
%   N11:1  PROC_OVERLAP_BUFFER  "STATE This holds the state during an overlap so the next state can be determined" %
%   N9:11  PROC_PURIFY_A  "STATE Process Purify A" %
%   N9:12  PROC_PURIFY_B  "STATE Process Purify B" %
%   N13:6/0  REGEN_COMPLETE  "STATUS Regen complete" %
%   N12:6/0  PURIFY_COMPLETE  "STATUS Purify complete" %

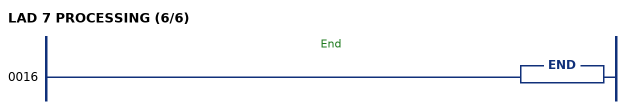
% Rung: 16 %
% End %
SOR END EOR

LADDER 8 "MANUAL_CTL"    % Runs the manual valve control %
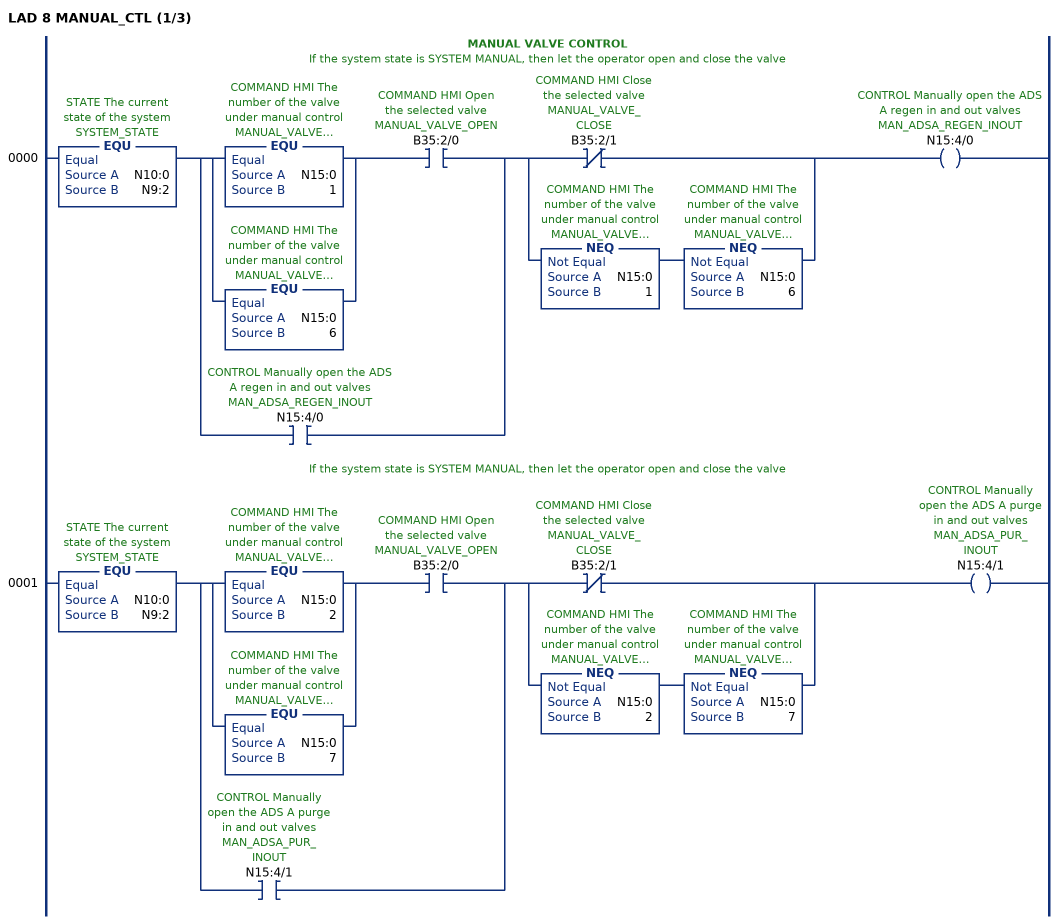
% Rung: 0 %
% TITLE: MANUAL VALVE CONTROL %
% If the system state is SYSTEM MANUAL, then let the operator open and close the valve %
SOR EQU N10:0 N9:2 BST BST EQU N15:0 1 NXB EQU N15:0 6 BND XIC B35:2/0 NXB XIC N15:4/0 BND BST XIO B35:2/1 NXB NEQ N15:0 1 NEQ N15:0 6 BND OTE N15:4/0 EOR
%   N10:0  SYSTEM_STATE  "STATE The current state of the system" %
%   N9:2  SYSTEM_MANUAL  "STATE System Manual" %
%   N15:0  MANUAL_VALVE_NUMBER  "COMMAND HMI The number of the valve under manual control" %
%   B35:2/0  MANUAL_VALVE_OPEN  "COMMAND HMI Open the selected valve" %
%   N15:4/0  MAN_ADSA_REGEN_INOUT  "CONTROL Manually open the ADS A regen in and out valves" %
%   B35:2/1  MANUAL_VALVE_CLOSE  "COMMAND HMI Close the selected valve" %
% Rung: 1 %
% If the system state is SYSTEM MANUAL, then let the operator open and close the valve %
SOR EQU N10:0 N9:2 BST BST EQU N15:0 2 NXB EQU N15:0 7 BND XIC B35:2/0 NXB XIC N15:4/1 BND BST XIO B35:2/1 NXB NEQ N15:0 2 NEQ N15:0 7 BND OTE N15:4/1 EOR
%   N10:0  SYSTEM_STATE  "STATE The current state of the system" %
%   N9:2  SYSTEM_MANUAL  "STATE System Manual" %
%   N15:0  MANUAL_VALVE_NUMBER  "COMMAND HMI The number of the valve under manual control" %
%   B35:2/0  MANUAL_VALVE_OPEN  "COMMAND HMI Open the selected valve" %
%   N15:4/1  MAN_ADSA_PUR_INOUT  "CONTROL Manually open the ADS A purge in and out valves" %
%   B35:2/1  MANUAL_VALVE_CLOSE  "COMMAND HMI Close the selected valve" %

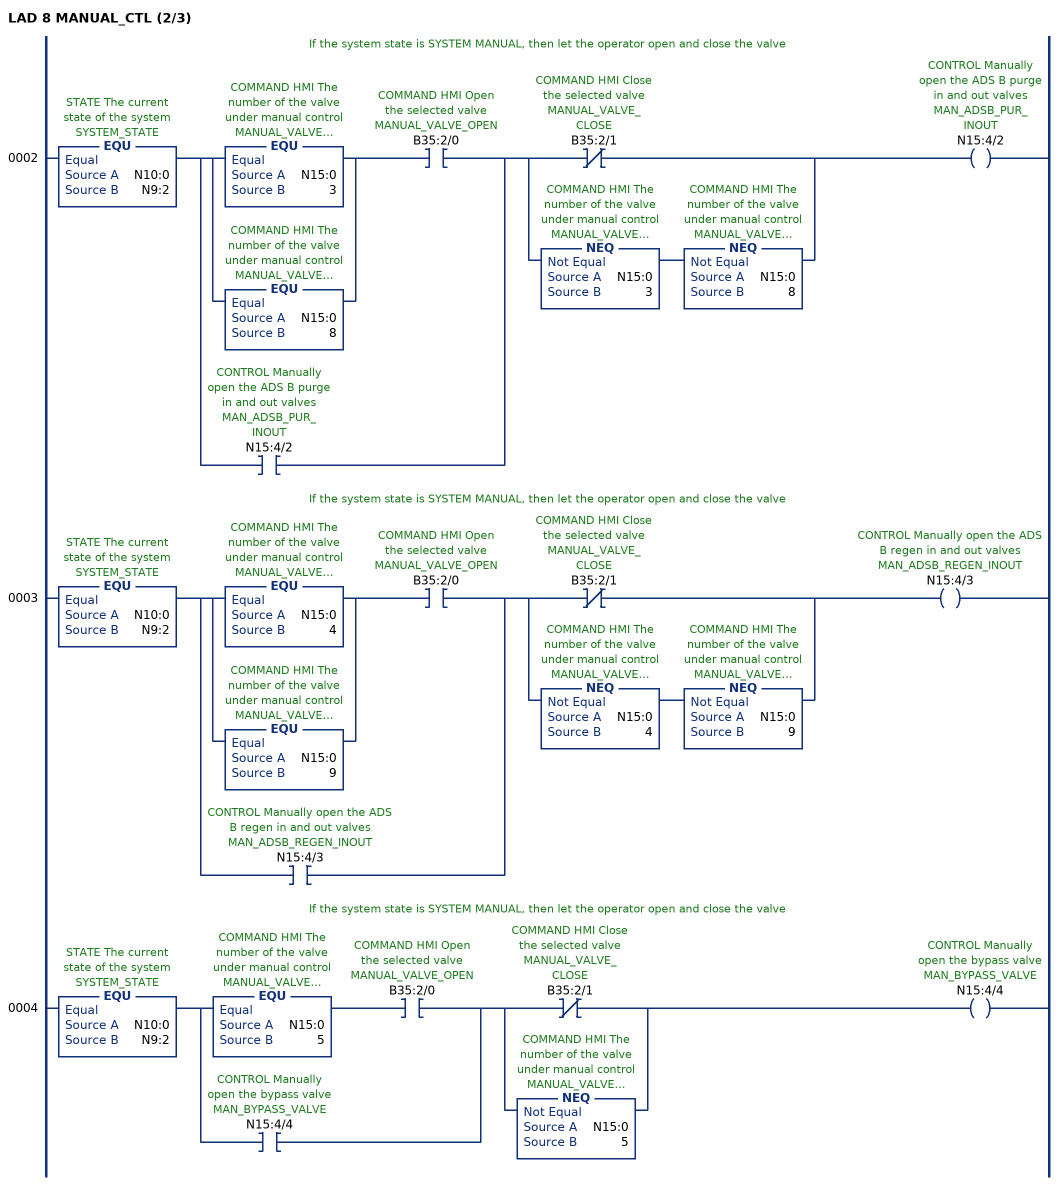
% Rung: 2 %
% If the system state is SYSTEM MANUAL, then let the operator open and close the valve %
SOR EQU N10:0 N9:2 BST BST EQU N15:0 3 NXB EQU N15:0 8 BND XIC B35:2/0 NXB XIC N15:4/2 BND BST XIO B35:2/1 NXB NEQ N15:0 3 NEQ N15:0 8 BND OTE N15:4/2 EOR
%   N10:0  SYSTEM_STATE  "STATE The current state of the system" %
%   N9:2  SYSTEM_MANUAL  "STATE System Manual" %
%   N15:0  MANUAL_VALVE_NUMBER  "COMMAND HMI The number of the valve under manual control" %
%   B35:2/0  MANUAL_VALVE_OPEN  "COMMAND HMI Open the selected valve" %
%   N15:4/2  MAN_ADSB_PUR_INOUT  "CONTROL Manually open the ADS B purge in and out valves" %
%   B35:2/1  MANUAL_VALVE_CLOSE  "COMMAND HMI Close the selected valve" %
% Rung: 3 %
% If the system state is SYSTEM MANUAL, then let the operator open and close the valve %
SOR EQU N10:0 N9:2 BST BST EQU N15:0 4 NXB EQU N15:0 9 BND XIC B35:2/0 NXB XIC N15:4/3 BND BST XIO B35:2/1 NXB NEQ N15:0 4 NEQ N15:0 9 BND OTE N15:4/3 EOR
%   N10:0  SYSTEM_STATE  "STATE The current state of the system" %
%   N9:2  SYSTEM_MANUAL  "STATE System Manual" %
%   N15:0  MANUAL_VALVE_NUMBER  "COMMAND HMI The number of the valve under manual control" %
%   B35:2/0  MANUAL_VALVE_OPEN  "COMMAND HMI Open the selected valve" %
%   N15:4/3  MAN_ADSB_REGEN_INOUT  "CONTROL Manually open the ADS B regen in and out valves" %
%   B35:2/1  MANUAL_VALVE_CLOSE  "COMMAND HMI Close the selected valve" %
% Rung: 4 %
% If the system state is SYSTEM MANUAL, then let the operator open and close the valve %
SOR EQU N10:0 N9:2 BST EQU N15:0 5 XIC B35:2/0 NXB XIC N15:4/4 BND BST XIO B35:2/1 NXB NEQ N15:0 5 BND OTE N15:4/4 EOR
%   N10:0  SYSTEM_STATE  "STATE The current state of the system" %
%   N9:2  SYSTEM_MANUAL  "STATE System Manual" %
%   N15:0  MANUAL_VALVE_NUMBER  "COMMAND HMI The number of the valve under manual control" %
%   B35:2/0  MANUAL_VALVE_OPEN  "COMMAND HMI Open the selected valve" %
%   N15:4/4  MAN_BYPASS_VALVE  "CONTROL Manually open the bypass valve" %
%   B35:2/1  MANUAL_VALVE_CLOSE  "COMMAND HMI Close the selected valve" %

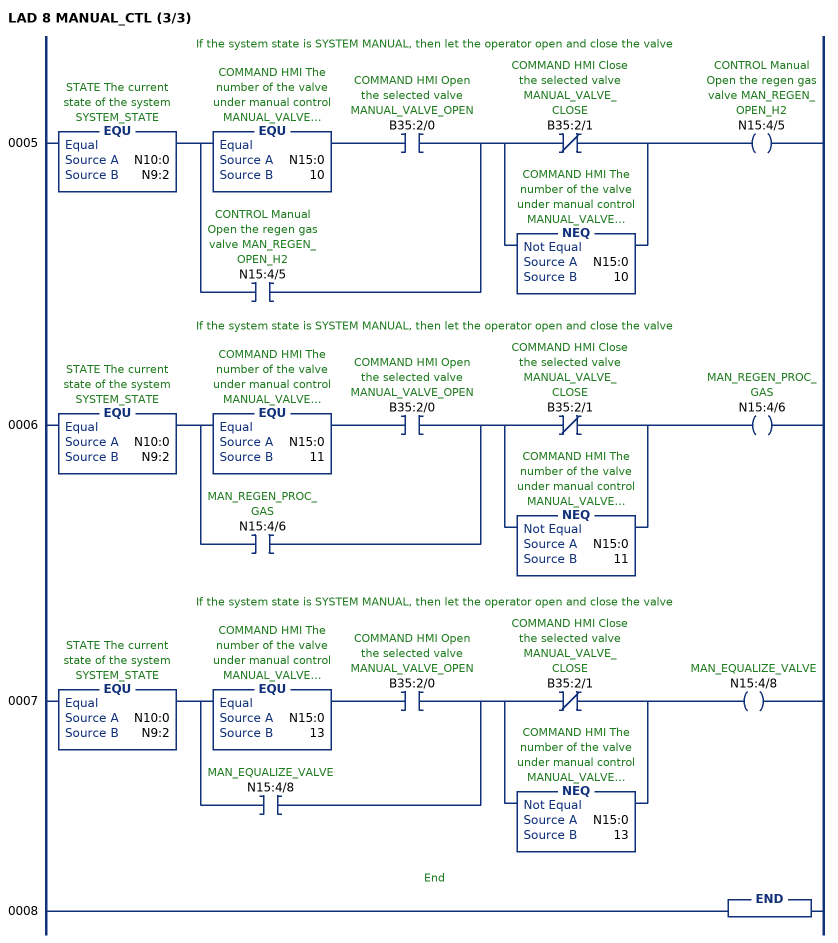
% Rung: 5 %
% If the system state is SYSTEM MANUAL, then let the operator open and close the valve %
SOR EQU N10:0 N9:2 BST EQU N15:0 10 XIC B35:2/0 NXB XIC N15:4/5 BND BST XIO B35:2/1 NXB NEQ N15:0 10 BND OTE N15:4/5 EOR
%   N10:0  SYSTEM_STATE  "STATE The current state of the system" %
%   N9:2  SYSTEM_MANUAL  "STATE System Manual" %
%   N15:0  MANUAL_VALVE_NUMBER  "COMMAND HMI The number of the valve under manual control" %
%   B35:2/0  MANUAL_VALVE_OPEN  "COMMAND HMI Open the selected valve" %
%   N15:4/5  MAN_REGEN_OPEN_H2  "CONTROL Manual Open the regen gas valve" %
%   B35:2/1  MANUAL_VALVE_CLOSE  "COMMAND HMI Close the selected valve" %
% Rung: 6 %
% If the system state is SYSTEM MANUAL, then let the operator open and close the valve %
SOR EQU N10:0 N9:2 BST EQU N15:0 11 XIC B35:2/0 NXB XIC N15:4/6 BND BST XIO B35:2/1 NXB NEQ N15:0 11 BND OTE N15:4/6 EOR
%   N10:0  SYSTEM_STATE  "STATE The current state of the system" %
%   N9:2  SYSTEM_MANUAL  "STATE System Manual" %
%   N15:0  MANUAL_VALVE_NUMBER  "COMMAND HMI The number of the valve under manual control" %
%   B35:2/0  MANUAL_VALVE_OPEN  "COMMAND HMI Open the selected valve" %
%   N15:4/6  MAN_REGEN_PROC_GAS %
%   B35:2/1  MANUAL_VALVE_CLOSE  "COMMAND HMI Close the selected valve" %
% Rung: 7 %
% If the system state is SYSTEM MANUAL, then let the operator open and close the valve %
SOR EQU N10:0 N9:2 BST EQU N15:0 13 XIC B35:2/0 NXB XIC N15:4/8 BND BST XIO B35:2/1 NXB NEQ N15:0 13 BND OTE N15:4/8 EOR
%   N10:0  SYSTEM_STATE  "STATE The current state of the system" %
%   N9:2  SYSTEM_MANUAL  "STATE System Manual" %
%   N15:0  MANUAL_VALVE_NUMBER  "COMMAND HMI The number of the valve under manual control" %
%   B35:2/0  MANUAL_VALVE_OPEN  "COMMAND HMI Open the selected valve" %
%   N15:4/8  MAN_EQUALIZE_VALVE %
%   B35:2/1  MANUAL_VALVE_CLOSE  "COMMAND HMI Close the selected valve" %
% Rung: 8 %
% End %
SOR END EOR

LADDER 10 "PURIFY"    % Operates the purify control %
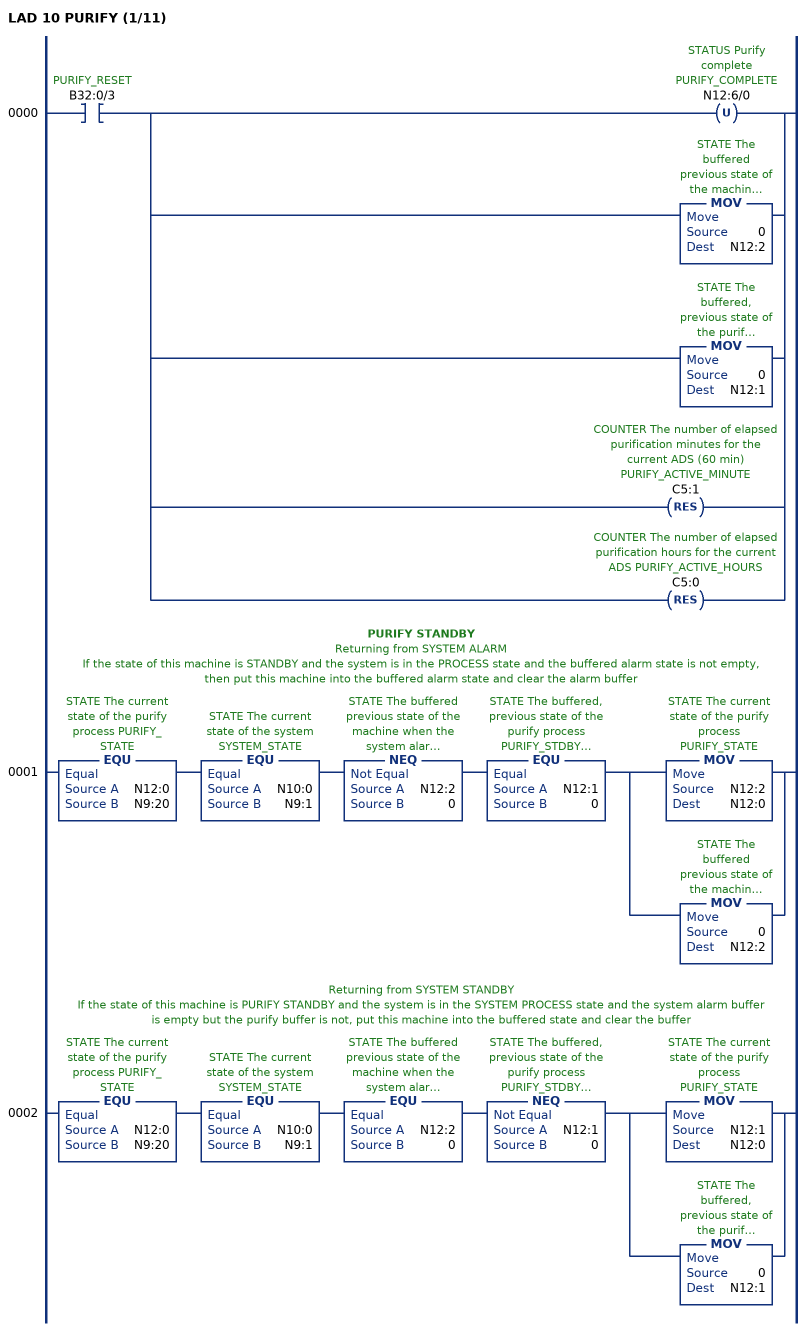
% Rung: 0 %
SOR XIC B32:0/3 BST OTU N12:6/0 NXB MOV 0 N12:2 NXB MOV 0 N12:1 NXB RES C5:1 NXB RES C5:0 BND EOR
%   B32:0/3  PURIFY_RESET %
%   N12:6/0  PURIFY_COMPLETE  "STATUS Purify complete" %
%   N12:2  PURIFY_ALARM_BUFFER  "STATE The buffered previous state of the machine when the system alarm occured" %
%   N12:1  PURIFY_STDBY_BUFFER  "STATE The buffered, previous state of the purify process" %
%   C5:1  PURIFY_ACTIVE_MINUTE  "COUNTER The number of elapsed purification minutes for the current ADS (60 min)" %
%   C5:0  PURIFY_ACTIVE_HOURS  "COUNTER The number of elapsed purification hours for the current ADS" %
% Rung: 1 %
% TITLE: PURIFY STANDBY %
% Returning from SYSTEM ALARM
% If the state of this machine is STANDBY and the system is in the PROCESS state and the buffered alarm state is not empty, then put this machine into the buffered alarm state and clear the alarm buffer %
SOR EQU N12:0 N9:20 EQU N10:0 N9:1 NEQ N12:2 0 EQU N12:1 0 BST MOV N12:2 N12:0 NXB MOV 0 N12:2 BND EOR
%   N12:0  PURIFY_STATE  "STATE The current state of the purify process" %
%   N9:20  PURIFY_STANDBY  "STATE Purify Standby" %
%   N10:0  SYSTEM_STATE  "STATE The current state of the system" %
%   N9:1  SYSTEM_PROCESS  "STATE System Process" %
%   N12:2  PURIFY_ALARM_BUFFER  "STATE The buffered previous state of the machine when the system alarm occured" %
%   N12:1  PURIFY_STDBY_BUFFER  "STATE The buffered, previous state of the purify process" %
% Rung: 2 %
% Returning from SYSTEM STANDBY
% If the state of this machine is PURIFY STANDBY and the system is in the SYSTEM PROCESS state and the system alarm buffer is empty but the purify buffer is not, put this machine into the buffered state and clear the buffer %
SOR EQU N12:0 N9:20 EQU N10:0 N9:1 EQU N12:2 0 NEQ N12:1 0 BST MOV N12:1 N12:0 NXB MOV 0 N12:1 BND EOR
%   N12:0  PURIFY_STATE  "STATE The current state of the purify process" %
%   N9:20  PURIFY_STANDBY  "STATE Purify Standby" %
%   N10:0  SYSTEM_STATE  "STATE The current state of the system" %
%   N9:1  SYSTEM_PROCESS  "STATE System Process" %
%   N12:2  PURIFY_ALARM_BUFFER  "STATE The buffered previous state of the machine when the system alarm occured" %
%   N12:1  PURIFY_STDBY_BUFFER  "STATE The buffered, previous state of the purify process" %

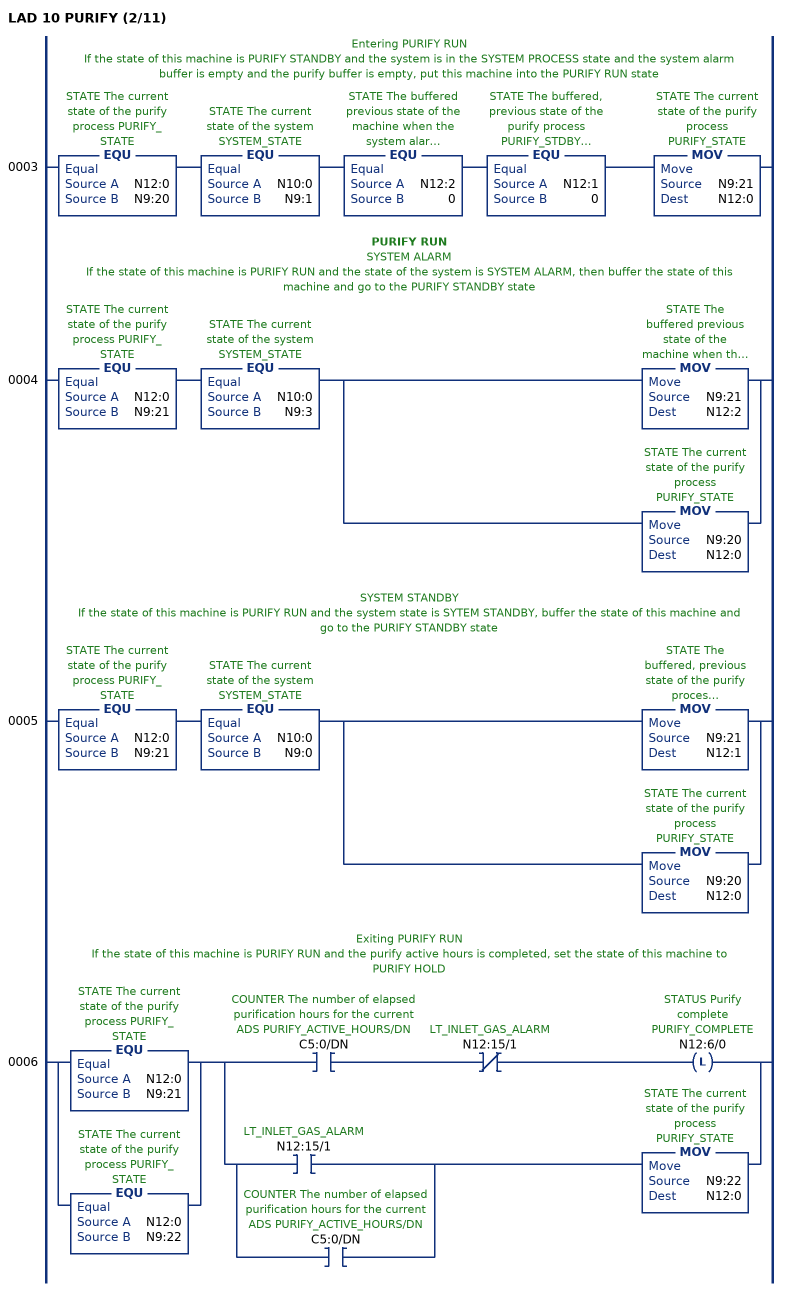
% Rung: 3 %
% Entering PURIFY RUN
% If the state of this machine is PURIFY STANDBY and the system is in the SYSTEM PROCESS state and the system alarm buffer is empty and the purify buffer is empty, put this machine into the PURIFY RUN state %
SOR EQU N12:0 N9:20 EQU N10:0 N9:1 EQU N12:2 0 EQU N12:1 0 MOV N9:21 N12:0 EOR
%   N12:0  PURIFY_STATE  "STATE The current state of the purify process" %
%   N9:20  PURIFY_STANDBY  "STATE Purify Standby" %
%   N10:0  SYSTEM_STATE  "STATE The current state of the system" %
%   N9:1  SYSTEM_PROCESS  "STATE System Process" %
%   N12:2  PURIFY_ALARM_BUFFER  "STATE The buffered previous state of the machine when the system alarm occured" %
%   N12:1  PURIFY_STDBY_BUFFER  "STATE The buffered, previous state of the purify process" %
%   N9:21  PURIFY_RUN  "STATE Purify running" %
% Rung: 4 %
% TITLE: PURIFY RUN %
% SYSTEM ALARM
% If the state of this machine is PURIFY RUN and the state of the system is SYSTEM ALARM, then buffer the state of this machine and go to the PURIFY STANDBY state %
SOR EQU N12:0 N9:21 EQU N10:0 N9:3 BST MOV N9:21 N12:2 NXB MOV N9:20 N12:0 BND EOR
%   N12:0  PURIFY_STATE  "STATE The current state of the purify process" %
%   N9:21  PURIFY_RUN  "STATE Purify running" %
%   N10:0  SYSTEM_STATE  "STATE The current state of the system" %
%   N9:3  SYSTEM_ALARM  "STATE System Alarm" %
%   N12:2  PURIFY_ALARM_BUFFER  "STATE The buffered previous state of the machine when the system alarm occured" %
%   N9:20  PURIFY_STANDBY  "STATE Purify Standby" %
% Rung: 5 %
% SYSTEM STANDBY
% If the state of this machine is PURIFY RUN and the system state is SYTEM STANDBY, buffer the state of this machine and go to the PURIFY STANDBY state %
SOR EQU N12:0 N9:21 EQU N10:0 N9:0 BST MOV N9:21 N12:1 NXB MOV N9:20 N12:0 BND EOR
%   N12:0  PURIFY_STATE  "STATE The current state of the purify process" %
%   N9:21  PURIFY_RUN  "STATE Purify running" %
%   N10:0  SYSTEM_STATE  "STATE The current state of the system" %
%   N9:0  SYSTEM_STANDBY  "STATE System Standby" %
%   N12:1  PURIFY_STDBY_BUFFER  "STATE The buffered, previous state of the purify process" %
%   N9:20  PURIFY_STANDBY  "STATE Purify Standby" %
% Rung: 6 %
% Exiting PURIFY RUN
% If the state of this machine is PURIFY RUN and the purify active hours is completed, set the state of this machine to PURIFY HOLD %
SOR BST EQU N12:0 N9:21 NXB EQU N12:0 N9:22 BND BST XIC C5:0/DN XIO N12:15/1 OTL N12:6/0 NXB BST XIC N12:15/1 NXB XIC C5:0/DN BND MOV N9:22 N12:0 BND EOR
%   N12:0  PURIFY_STATE  "STATE The current state of the purify process" %
%   N9:21  PURIFY_RUN  "STATE Purify running" %
%   N9:22  PURIFY_HOLD  "STATE Purify Hold" %
%   C5:0  PURIFY_ACTIVE_HOURS  "COUNTER The number of elapsed purification hours for the current ADS" %
%   N12:15/1  LT_INLET_GAS_ALARM %
%   N12:6/0  PURIFY_COMPLETE  "STATUS Purify complete" %

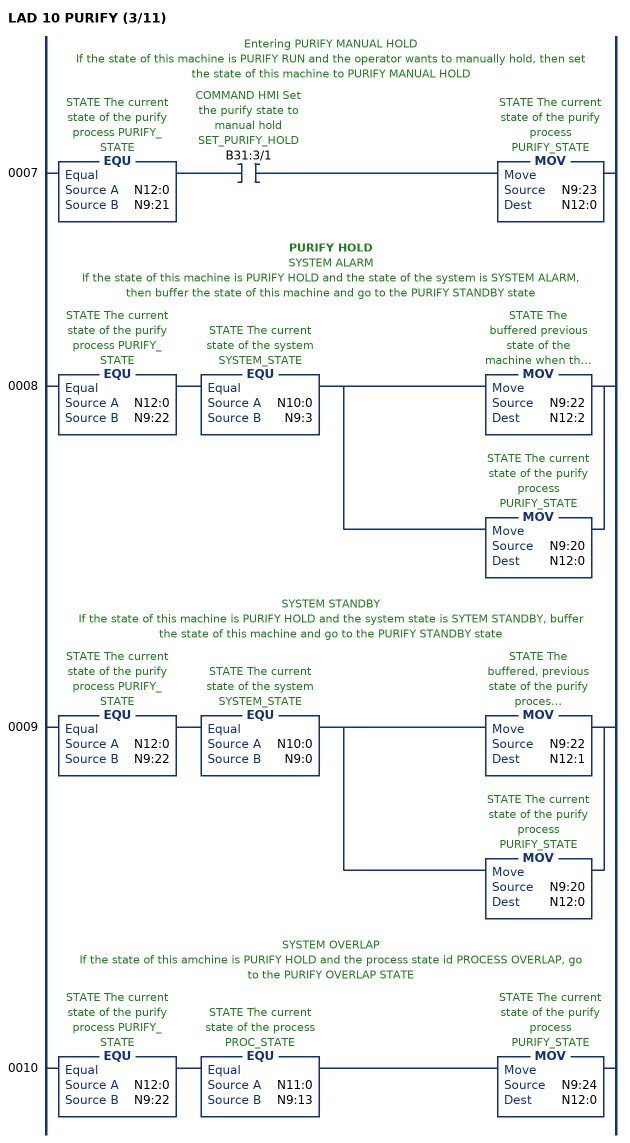
% Rung: 7 %
% Entering PURIFY MANUAL HOLD
% If the state of this machine is PURIFY RUN and the operator wants to manually hold, then set the state of this machine to PURIFY MANUAL HOLD %
SOR EQU N12:0 N9:21 XIC B31:3/1 MOV N9:23 N12:0 EOR
%   N12:0  PURIFY_STATE  "STATE The current state of the purify process" %
%   N9:21  PURIFY_RUN  "STATE Purify running" %
%   B31:3/1  SET_PURIFY_HOLD  "COMMAND HMI Set the purify state to manual hold" %
%   N9:23  PURIFY_MANUAL_HOLD  "STATE Purify Manual Hold" %
% Rung: 8 %
% TITLE: PURIFY HOLD %
% SYSTEM ALARM
% If the state of this machine is PURIFY HOLD and the state of the system is SYSTEM ALARM, then buffer the state of this machine and go to the PURIFY STANDBY state %
SOR EQU N12:0 N9:22 EQU N10:0 N9:3 BST MOV N9:22 N12:2 NXB MOV N9:20 N12:0 BND EOR
%   N12:0  PURIFY_STATE  "STATE The current state of the purify process" %
%   N9:22  PURIFY_HOLD  "STATE Purify Hold" %
%   N10:0  SYSTEM_STATE  "STATE The current state of the system" %
%   N9:3  SYSTEM_ALARM  "STATE System Alarm" %
%   N12:2  PURIFY_ALARM_BUFFER  "STATE The buffered previous state of the machine when the system alarm occured" %
%   N9:20  PURIFY_STANDBY  "STATE Purify Standby" %
% Rung: 9 %
% SYSTEM STANDBY
% If the state of this machine is PURIFY HOLD and the system state is SYTEM STANDBY, buffer the state of this machine and go to the PURIFY STANDBY state %
SOR EQU N12:0 N9:22 EQU N10:0 N9:0 BST MOV N9:22 N12:1 NXB MOV N9:20 N12:0 BND EOR
%   N12:0  PURIFY_STATE  "STATE The current state of the purify process" %
%   N9:22  PURIFY_HOLD  "STATE Purify Hold" %
%   N10:0  SYSTEM_STATE  "STATE The current state of the system" %
%   N9:0  SYSTEM_STANDBY  "STATE System Standby" %
%   N12:1  PURIFY_STDBY_BUFFER  "STATE The buffered, previous state of the purify process" %
%   N9:20  PURIFY_STANDBY  "STATE Purify Standby" %
% Rung: 10 %
% SYSTEM OVERLAP
% If the state of this amchine is PURIFY HOLD and the process state id PROCESS OVERLAP, go to the PURIFY OVERLAP STATE %
SOR EQU N12:0 N9:22 EQU N11:0 N9:13 MOV N9:24 N12:0 EOR
%   N12:0  PURIFY_STATE  "STATE The current state of the purify process" %
%   N9:22  PURIFY_HOLD  "STATE Purify Hold" %
%   N11:0  PROC_STATE  "STATE The current state of the process" %
%   N9:13  PROC_OVERLAP  "STATE Process Purify Overlap" %
%   N9:24  PURIFY_OVERLAP  "STATE Puriify Overlap" %

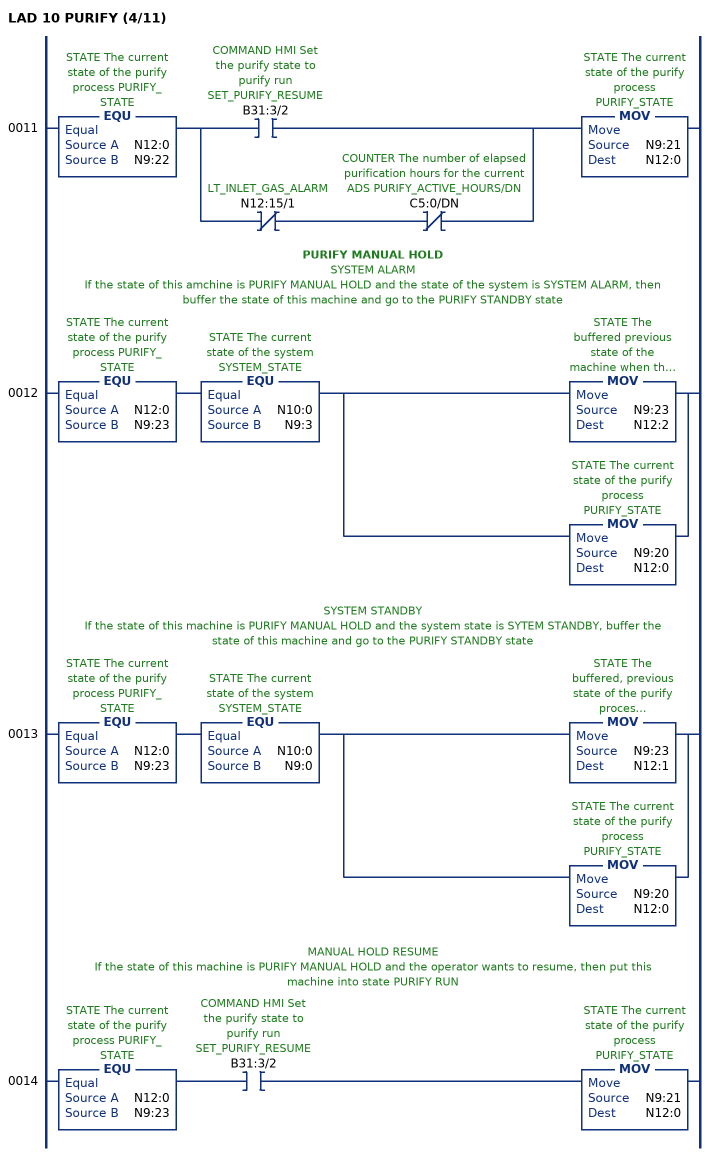
% Rung: 11 %
SOR EQU N12:0 N9:22 BST XIC B31:3/2 NXB XIO N12:15/1 XIO C5:0/DN BND MOV N9:21 N12:0 EOR
%   N12:0  PURIFY_STATE  "STATE The current state of the purify process" %
%   N9:22  PURIFY_HOLD  "STATE Purify Hold" %
%   B31:3/2  SET_PURIFY_RESUME  "COMMAND HMI Set the purify state to purify run" %
%   N12:15/1  LT_INLET_GAS_ALARM %
%   C5:0  PURIFY_ACTIVE_HOURS  "COUNTER The number of elapsed purification hours for the current ADS" %
%   N9:21  PURIFY_RUN  "STATE Purify running" %
% Rung: 12 %
% TITLE: PURIFY MANUAL HOLD %
% SYSTEM ALARM
% If the state of this amchine is PURIFY MANUAL HOLD and the state of the system is SYSTEM ALARM, then buffer the state of this machine and go to the PURIFY STANDBY state %
SOR EQU N12:0 N9:23 EQU N10:0 N9:3 BST MOV N9:23 N12:2 NXB MOV N9:20 N12:0 BND EOR
%   N12:0  PURIFY_STATE  "STATE The current state of the purify process" %
%   N9:23  PURIFY_MANUAL_HOLD  "STATE Purify Manual Hold" %
%   N10:0  SYSTEM_STATE  "STATE The current state of the system" %
%   N9:3  SYSTEM_ALARM  "STATE System Alarm" %
%   N12:2  PURIFY_ALARM_BUFFER  "STATE The buffered previous state of the machine when the system alarm occured" %
%   N9:20  PURIFY_STANDBY  "STATE Purify Standby" %
% Rung: 13 %
% SYSTEM STANDBY
% If the state of this machine is PURIFY MANUAL HOLD and the system state is SYTEM STANDBY, buffer the state of this machine and go to the PURIFY STANDBY state %
SOR EQU N12:0 N9:23 EQU N10:0 N9:0 BST MOV N9:23 N12:1 NXB MOV N9:20 N12:0 BND EOR
%   N12:0  PURIFY_STATE  "STATE The current state of the purify process" %
%   N9:23  PURIFY_MANUAL_HOLD  "STATE Purify Manual Hold" %
%   N10:0  SYSTEM_STATE  "STATE The current state of the system" %
%   N9:0  SYSTEM_STANDBY  "STATE System Standby" %
%   N12:1  PURIFY_STDBY_BUFFER  "STATE The buffered, previous state of the purify process" %
%   N9:20  PURIFY_STANDBY  "STATE Purify Standby" %
% Rung: 14 %
% MANUAL HOLD RESUME
% If the state of this machine is PURIFY MANUAL HOLD and the operator wants to resume, then put this machine into state PURIFY RUN %
SOR EQU N12:0 N9:23 XIC B31:3/2 MOV N9:21 N12:0 EOR
%   N12:0  PURIFY_STATE  "STATE The current state of the purify process" %
%   N9:23  PURIFY_MANUAL_HOLD  "STATE Purify Manual Hold" %
%   B31:3/2  SET_PURIFY_RESUME  "COMMAND HMI Set the purify state to purify run" %
%   N9:21  PURIFY_RUN  "STATE Purify running" %

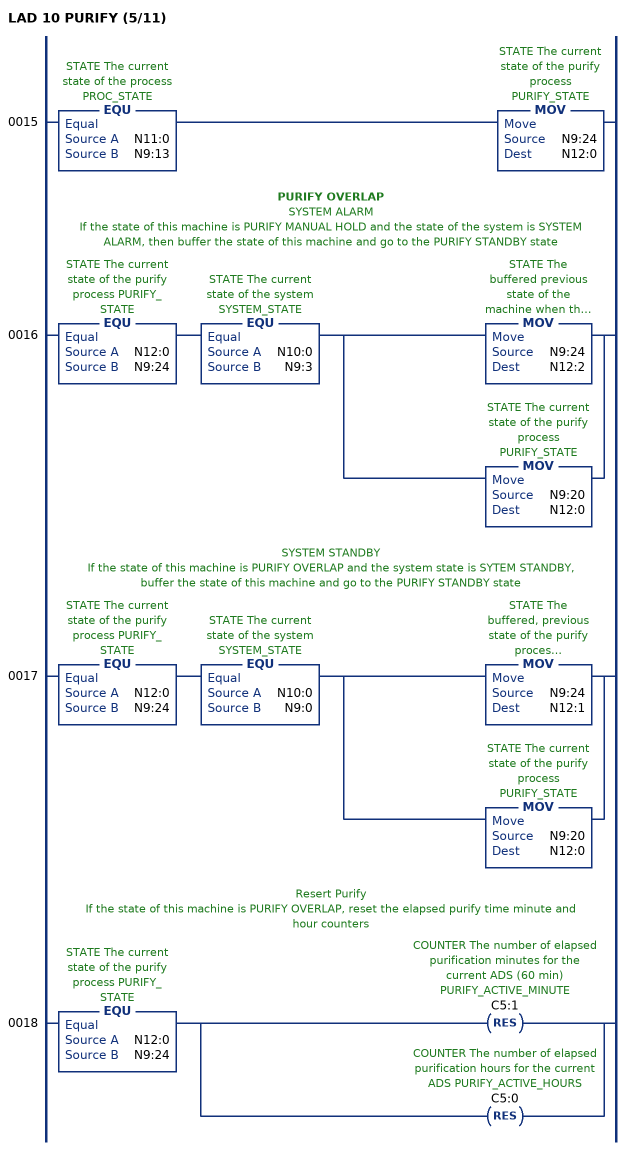
% Rung: 15 %
SOR EQU N11:0 N9:13 MOV N9:24 N12:0 EOR
%   N11:0  PROC_STATE  "STATE The current state of the process" %
%   N9:13  PROC_OVERLAP  "STATE Process Purify Overlap" %
%   N9:24  PURIFY_OVERLAP  "STATE Puriify Overlap" %
%   N12:0  PURIFY_STATE  "STATE The current state of the purify process" %
% Rung: 16 %
% TITLE: PURIFY OVERLAP %
% SYSTEM ALARM
% If the state of this machine is PURIFY MANUAL HOLD and the state of the system is SYSTEM ALARM, then buffer the state of this machine and go to the PURIFY STANDBY state %
SOR EQU N12:0 N9:24 EQU N10:0 N9:3 BST MOV N9:24 N12:2 NXB MOV N9:20 N12:0 BND EOR
%   N12:0  PURIFY_STATE  "STATE The current state of the purify process" %
%   N9:24  PURIFY_OVERLAP  "STATE Puriify Overlap" %
%   N10:0  SYSTEM_STATE  "STATE The current state of the system" %
%   N9:3  SYSTEM_ALARM  "STATE System Alarm" %
%   N12:2  PURIFY_ALARM_BUFFER  "STATE The buffered previous state of the machine when the system alarm occured" %
%   N9:20  PURIFY_STANDBY  "STATE Purify Standby" %
% Rung: 17 %
% SYSTEM STANDBY
% If the state of this machine is PURIFY OVERLAP and the system state is SYTEM STANDBY, buffer the state of this machine and go to the PURIFY STANDBY state %
SOR EQU N12:0 N9:24 EQU N10:0 N9:0 BST MOV N9:24 N12:1 NXB MOV N9:20 N12:0 BND EOR
%   N12:0  PURIFY_STATE  "STATE The current state of the purify process" %
%   N9:24  PURIFY_OVERLAP  "STATE Puriify Overlap" %
%   N10:0  SYSTEM_STATE  "STATE The current state of the system" %
%   N9:0  SYSTEM_STANDBY  "STATE System Standby" %
%   N12:1  PURIFY_STDBY_BUFFER  "STATE The buffered, previous state of the purify process" %
%   N9:20  PURIFY_STANDBY  "STATE Purify Standby" %
% Rung: 18 %
% Resert Purify
% If the state of this machine is PURIFY OVERLAP, reset the elapsed purify time minute and hour counters %
SOR EQU N12:0 N9:24 BST RES C5:1 NXB RES C5:0 BND EOR
%   N12:0  PURIFY_STATE  "STATE The current state of the purify process" %
%   N9:24  PURIFY_OVERLAP  "STATE Puriify Overlap" %
%   C5:1  PURIFY_ACTIVE_MINUTE  "COUNTER The number of elapsed purification minutes for the current ADS (60 min)" %
%   C5:0  PURIFY_ACTIVE_HOURS  "COUNTER The number of elapsed purification hours for the current ADS" %

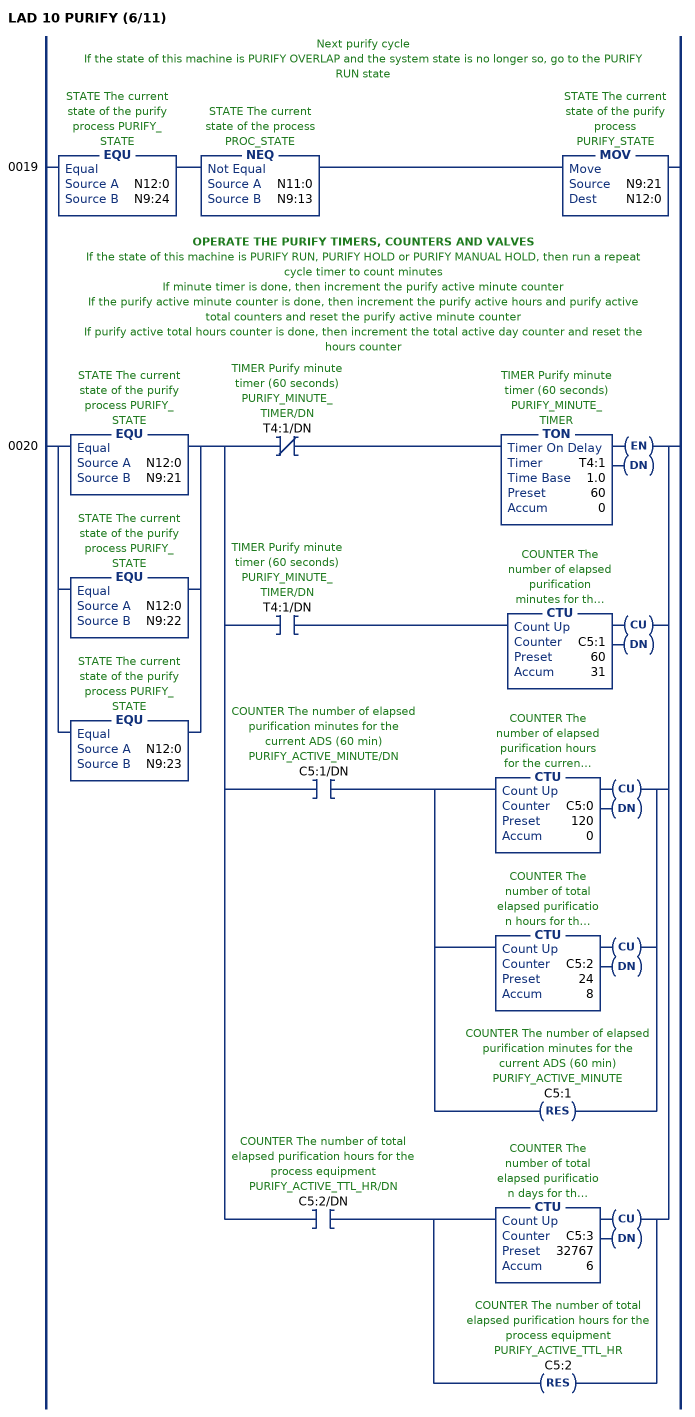
% Rung: 19 %
% Next purify cycle
% If the state of this machine is PURIFY OVERLAP and the system state is no longer so, go to the PURIFY RUN state %
SOR EQU N12:0 N9:24 NEQ N11:0 N9:13 MOV N9:21 N12:0 EOR
%   N12:0  PURIFY_STATE  "STATE The current state of the purify process" %
%   N9:24  PURIFY_OVERLAP  "STATE Puriify Overlap" %
%   N11:0  PROC_STATE  "STATE The current state of the process" %
%   N9:13  PROC_OVERLAP  "STATE Process Purify Overlap" %
%   N9:21  PURIFY_RUN  "STATE Purify running" %
% Rung: 20 %
% TITLE: OPERATE THE PURIFY TIMERS, COUNTERS AND VALVES %
% If the state of this machine is PURIFY RUN, PURIFY HOLD or PURIFY MANUAL HOLD, then run a repeat cycle timer to count minutes
% If minute timer is done, then increment the purify active minute counter
% If the purify active minute counter is done, then increment the purify active hours and purify active total counters and reset the purify active minute counter
% If purify active total hours counter is done, then increment the total active day counter and reset the hours counter %
SOR BST EQU N12:0 N9:21 NXB EQU N12:0 N9:22 NXB EQU N12:0 N9:23 BND BST XIO T4:1/DN TON T4:1 1.0 60 0 NXB XIC T4:1/DN CTU C5:1 60 31 NXB XIC C5:1/DN BST CTU C5:0 120 0 NXB CTU C5:2 24 8 NXB RES C5:1 BND NXB XIC C5:2/DN BST CTU C5:3 32767 6 NXB RES C5:2 BND BND EOR
%   N12:0  PURIFY_STATE  "STATE The current state of the purify process" %
%   N9:21  PURIFY_RUN  "STATE Purify running" %
%   N9:22  PURIFY_HOLD  "STATE Purify Hold" %
%   N9:23  PURIFY_MANUAL_HOLD  "STATE Purify Manual Hold" %
%   T4:1  PURIFY_MINUTE_TIMER  "TIMER Purify minute timer (60 seconds)" %
%   C5:1  PURIFY_ACTIVE_MINUTE  "COUNTER The number of elapsed purification minutes for the current ADS (60 min)" %
%   C5:0  PURIFY_ACTIVE_HOURS  "COUNTER The number of elapsed purification hours for the current ADS" %
%   C5:2  PURIFY_ACTIVE_TTL_HR  "COUNTER The number of total elapsed purification hours for the process equipment" %
%   C5:3  PURIFY_ACTIVE_TTL_DY  "COUNTER The number of total elapsed purification days for the process equipment" %

